	170: //Set the target power to each device
		//Batterys or battery inverters
		//Batterys are only a "normal" Device, when the self consumption mode is active.
		IF eOperationMode = E_OperatingMode_EMS.eSelfConsumption THEN 
			FOR liLPSetPercentPower := 1 TO Constants_Energy.diMaxNumberOfBatteryInverters BY 1 DO
				IF bSurplusAvailable AND Lynus_Standards.GVL_Energy.stDataOfBatteryInverters[diNrOfEMS_OUT,liLPSetPercentPower].byPriority = bySmGrActiveCommonPrio AND Lynus_Standards.GVL_Energy.stDataOfBatteryInverters[diNrOfEMS_OUT,liLPSetPercentPower].rTargetPowerEMS > -100 THEN 
					Lynus_Standards.GVL_Energy.stDataOfBatteryInverters[diNrOfEMS_OUT,liLPSetPercentPower].rTargetPowerEMS := Lynus_Standards.GVL_Energy.stDataOfBatteryInverters[diNrOfEMS_OUT,liLPSetPercentPower].rTargetPowerEMS - rValuePercentToControllableDevices; 
				END_IF
				IF bSurplusAvailable AND Lynus_Standards.GVL_Energy.stDataOfBatteryInverters[diNrOfEMS_OUT,liLPSetPercentPower].rTargetPowerEMS < -100 THEN 
					Lynus_Standards.GVL_Energy.stDataOfBatteryInverters[diNrOfEMS_OUT,liLPSetPercentPower].rTargetPowerEMS := -100; 
				END_IF 
				IF NOT bSurplusAvailable AND Lynus_Standards.GVL_Energy.stDataOfBatteryInverters[diNrOfEMS_OUT,liLPSetPercentPower].byPriority = bySmGrActiveCommonPrio AND Lynus_Standards.GVL_Energy.stDataOfBatteryInverters[diNrOfEMS_OUT,liLPSetPercentPower].rTargetPowerEMS < 0 THEN 
					Lynus_Standards.GVL_Energy.stDataOfBatteryInverters[diNrOfEMS_OUT,liLPSetPercentPower].rTargetPowerEMS := Lynus_Standards.GVL_Energy.stDataOfBatteryInverters[diNrOfEMS_OUT,liLPSetPercentPower].rTargetPowerEMS + rValuePercentToControllableDevices; 
				END_IF
				IF NOT bSurplusAvailable AND Lynus_Standards.GVL_Energy.stDataOfBatteryInverters[diNrOfEMS_OUT,liLPSetPercentPower].rTargetPowerEMS > 0 THEN 
					Lynus_Standards.GVL_Energy.stDataOfBatteryInverters[diNrOfEMS_OUT,liLPSetPercentPower].rTargetPowerEMS := 0; 
				END_IF
				//Power Data is Missing
				IF bMissingPowerData AND Lynus_Standards.GVL_Energy.stDataOfBatteryInverters[diNrOfEMS_OUT,liLPSetPercentPower].byPriority = bySmGrActiveCommonPrio THEN 
					Lynus_Standards.GVL_Energy.stDataOfBatteryInverters[diNrOfEMS_OUT,liLPSetPercentPower].rTargetPowerEMS := 0;	
				END_IF 
				//Limit
				Lynus_Standards.GVL_Energy.stDataOfBatteryInverters[diNrOfEMS_OUT,liLPSetPercentPower].rTargetPowerEMS := LIMIT(-100,Lynus_Standards.GVL_Energy.stDataOfBatteryInverters[diNrOfEMS_OUT,liLPSetPercentPower].rTargetPowerEMS,100);	
			END_FOR
		END_IF
		//Heating pumps
		IF arrActualStepInTurn[1] >= 1 AND arrActualStepInTurn[1] <= 2 THEN
			FOR liLPSetPercentPower := 1 TO Constants_Energy.diMaxNumberOfHeatingPumps BY 1 DO
				//On/Off
				IF bSurplusAvailable AND Lynus_Standards.GVL_Energy.stDataHeatingPumps[diNrOfEMS_OUT,liLPSetPercentPower].byPriority = bySmGrActiveCommonPrio AND Lynus_Standards.GVL_Energy.stDataHeatingPumps[diNrOfEMS_OUT,liLPSetPercentPower].arrTargetPowerEMS[arrActualStepInTurn[1]] < 100 AND NOT 
				Lynus_Standards.GVL_Energy.stDataHeatingPumps[diNrOfEMS_OUT,liLPSetPercentPower].bIsControllable AND NOT Lynus_Standards.GVL_Energy.stDataHeatingPumps[diNrOfEMS_OUT,liLPSetPercentPower].bIsStepSwitched THEN
					Lynus_Standards.GVL_Energy.stDataHeatingPumps[diNrOfEMS_OUT,liLPSetPercentPower].arrTargetPowerEMS[arrActualStepInTurn[1]] := rValuePercentToStepSwitchedDevices; 
				END_IF
				//Controllable linear
				IF bSurplusAvailable AND Lynus_Standards.GVL_Energy.stDataHeatingPumps[diNrOfEMS_OUT,liLPSetPercentPower].byPriority = bySmGrActiveCommonPrio AND Lynus_Standards.GVL_Energy.stDataHeatingPumps[diNrOfEMS_OUT,liLPSetPercentPower].arrTargetPowerEMS[arrActualStepInTurn[1]] < 100 AND 
				Lynus_Standards.GVL_Energy.stDataHeatingPumps[diNrOfEMS_OUT,liLPSetPercentPower].bIsControllable AND NOT Lynus_Standards.GVL_Energy.stDataHeatingPumps[diNrOfEMS_OUT,liLPSetPercentPower].bIsStepSwitched THEN
					Lynus_Standards.GVL_Energy.stDataHeatingPumps[diNrOfEMS_OUT,liLPSetPercentPower].arrTargetPowerEMS[arrActualStepInTurn[1]] := Lynus_Standards.GVL_Energy.stDataHeatingPumps[diNrOfEMS_OUT,liLPSetPercentPower].arrTargetPowerEMS[arrActualStepInTurn[1]] + rValuePercentToControllableDevices; 
				END_IF
				//Step switched
				IF bSurplusAvailable AND Lynus_Standards.GVL_Energy.stDataHeatingPumps[diNrOfEMS_OUT,liLPSetPercentPower].byPriority = bySmGrActiveCommonPrio AND Lynus_Standards.GVL_Energy.stDataHeatingPumps[diNrOfEMS_OUT,liLPSetPercentPower].arrTargetPowerEMS[arrActualStepInTurn[1]] < 100 AND 
				Lynus_Standards.GVL_Energy.stDataHeatingPumps[diNrOfEMS_OUT,liLPSetPercentPower].bIsControllable AND Lynus_Standards.GVL_Energy.stDataHeatingPumps[diNrOfEMS_OUT,liLPSetPercentPower].bIsStepSwitched THEN
					Lynus_Standards.GVL_Energy.stDataHeatingPumps[diNrOfEMS_OUT,liLPSetPercentPower].arrTargetPowerEMS[arrActualStepInTurn[1]] := rValuePercentToStepSwitchedDevices; 
				END_IF
				IF bSurplusAvailable AND Lynus_Standards.GVL_Energy.stDataHeatingPumps[diNrOfEMS_OUT,liLPSetPercentPower].arrTargetPowerEMS[arrActualStepInTurn[1]] > 100 THEN 
					Lynus_Standards.GVL_Energy.stDataHeatingPumps[diNrOfEMS_OUT,liLPSetPercentPower].arrTargetPowerEMS[arrActualStepInTurn[1]] := 100; 
				END_IF 
				//On/Off
				IF NOT bSurplusAvailable AND Lynus_Standards.GVL_Energy.stDataHeatingPumps[diNrOfEMS_OUT,liLPSetPercentPower].byPriority = bySmGrActiveCommonPrio AND Lynus_Standards.GVL_Energy.stDataHeatingPumps[diNrOfEMS_OUT,liLPSetPercentPower].arrTargetPowerEMS[arrActualStepInTurn[1]] > 0 AND NOT 
				Lynus_Standards.GVL_Energy.stDataHeatingPumps[diNrOfEMS_OUT,liLPSetPercentPower].bIsControllable AND NOT Lynus_Standards.GVL_Energy.stDataHeatingPumps[diNrOfEMS_OUT,liLPSetPercentPower].bIsStepSwitched THEN
					Lynus_Standards.GVL_Energy.stDataHeatingPumps[diNrOfEMS_OUT,liLPSetPercentPower].arrTargetPowerEMS[arrActualStepInTurn[1]] := rValuePercentToStepSwitchedDevices; 
				END_IF
				//Controllable linear
				IF NOT bSurplusAvailable AND Lynus_Standards.GVL_Energy.stDataHeatingPumps[diNrOfEMS_OUT,liLPSetPercentPower].byPriority = bySmGrActiveCommonPrio AND Lynus_Standards.GVL_Energy.stDataHeatingPumps[diNrOfEMS_OUT,liLPSetPercentPower].arrTargetPowerEMS[arrActualStepInTurn[1]] > 0 AND 
				Lynus_Standards.GVL_Energy.stDataHeatingPumps[diNrOfEMS_OUT,liLPSetPercentPower].bIsControllable AND NOT Lynus_Standards.GVL_Energy.stDataHeatingPumps[diNrOfEMS_OUT,liLPSetPercentPower].bIsStepSwitched THEN
					Lynus_Standards.GVL_Energy.stDataHeatingPumps[diNrOfEMS_OUT,liLPSetPercentPower].arrTargetPowerEMS[arrActualStepInTurn[1]] := Lynus_Standards.GVL_Energy.stDataHeatingPumps[diNrOfEMS_OUT,liLPSetPercentPower].arrTargetPowerEMS[arrActualStepInTurn[1]] - rValuePercentToControllableDevices; 
				END_IF
				//Step switched
				IF NOT bSurplusAvailable AND Lynus_Standards.GVL_Energy.stDataHeatingPumps[diNrOfEMS_OUT,liLPSetPercentPower].byPriority = bySmGrActiveCommonPrio AND Lynus_Standards.GVL_Energy.stDataHeatingPumps[diNrOfEMS_OUT,liLPSetPercentPower].arrTargetPowerEMS[arrActualStepInTurn[1]] > 0 AND 
				Lynus_Standards.GVL_Energy.stDataHeatingPumps[diNrOfEMS_OUT,liLPSetPercentPower].bIsControllable AND Lynus_Standards.GVL_Energy.stDataHeatingPumps[diNrOfEMS_OUT,liLPSetPercentPower].bIsStepSwitched THEN
					Lynus_Standards.GVL_Energy.stDataHeatingPumps[diNrOfEMS_OUT,liLPSetPercentPower].arrTargetPowerEMS[arrActualStepInTurn[1]] := rValuePercentToStepSwitchedDevices; 
				END_IF
				IF NOT bSurplusAvailable AND Lynus_Standards.GVL_Energy.stDataHeatingPumps[diNrOfEMS_OUT,liLPSetPercentPower].arrTargetPowerEMS[arrActualStepInTurn[1]] < 0 THEN 
					Lynus_Standards.GVL_Energy.stDataHeatingPumps[diNrOfEMS_OUT,liLPSetPercentPower].arrTargetPowerEMS[arrActualStepInTurn[1]] := 0; 
				END_IF
				//Limit
				Lynus_Standards.GVL_Energy.stDataHeatingPumps[diNrOfEMS_OUT,liLPSetPercentPower].arrTargetPowerEMS[arrActualStepInTurn[1]] := LIMIT(0,Lynus_Standards.GVL_Energy.stDataHeatingPumps[diNrOfEMS_OUT,liLPSetPercentPower].arrTargetPowerEMS[arrActualStepInTurn[1]],100);
			END_FOR
		END_IF
		//electric heating element
		IF arrActualStepInTurn[2] >= 1 AND arrActualStepInTurn[2] <= 10 THEN
			FOR liLPSetPercentPower := 1 TO Constants_Energy.diMaxNumberOfElectricHeatingElements BY 1 DO
				//On/Off
				IF bSurplusAvailable AND Lynus_Standards.GVL_Energy.stDataElectricHeatingElements[diNrOfEMS_OUT,liLPSetPercentPower].byPriority = bySmGrActiveCommonPrio AND Lynus_Standards.GVL_Energy.stDataElectricHeatingElements[diNrOfEMS_OUT,liLPSetPercentPower].arrTargetPowerEMS[arrActualStepInTurn[2]] < 100 AND NOT
				Lynus_Standards.GVL_Energy.stDataElectricHeatingElements[diNrOfEMS_OUT,liLPSetPercentPower].bIsControllable AND NOT Lynus_Standards.GVL_Energy.stDataElectricHeatingElements[diNrOfEMS_OUT,liLPSetPercentPower].bIsStepSwitched THEN
					Lynus_Standards.GVL_Energy.stDataElectricHeatingElements[diNrOfEMS_OUT,liLPSetPercentPower].arrTargetPowerEMS[arrActualStepInTurn[2]] := rValuePercentToStepSwitchedDevices;
				END_IF
				//Controllable linear
				IF bSurplusAvailable AND Lynus_Standards.GVL_Energy.stDataElectricHeatingElements[diNrOfEMS_OUT,liLPSetPercentPower].byPriority = bySmGrActiveCommonPrio AND Lynus_Standards.GVL_Energy.stDataElectricHeatingElements[diNrOfEMS_OUT,liLPSetPercentPower].arrTargetPowerEMS[arrActualStepInTurn[2]] < 100 AND
				Lynus_Standards.GVL_Energy.stDataElectricHeatingElements[diNrOfEMS_OUT,liLPSetPercentPower].bIsControllable AND NOT Lynus_Standards.GVL_Energy.stDataElectricHeatingElements[diNrOfEMS_OUT,liLPSetPercentPower].bIsStepSwitched THEN
					Lynus_Standards.GVL_Energy.stDataElectricHeatingElements[diNrOfEMS_OUT,liLPSetPercentPower].arrTargetPowerEMS[arrActualStepInTurn[2]] := Lynus_Standards.GVL_Energy.stDataElectricHeatingElements[diNrOfEMS_OUT,liLPSetPercentPower].arrTargetPowerEMS[arrActualStepInTurn[2]] + rValuePercentToControllableDevices;
				END_IF
				//Step switched
				IF bSurplusAvailable AND Lynus_Standards.GVL_Energy.stDataElectricHeatingElements[diNrOfEMS_OUT,liLPSetPercentPower].byPriority = bySmGrActiveCommonPrio AND Lynus_Standards.GVL_Energy.stDataElectricHeatingElements[diNrOfEMS_OUT,liLPSetPercentPower].arrTargetPowerEMS[arrActualStepInTurn[2]] < 100 AND
				Lynus_Standards.GVL_Energy.stDataElectricHeatingElements[diNrOfEMS_OUT,liLPSetPercentPower].bIsControllable AND Lynus_Standards.GVL_Energy.stDataElectricHeatingElements[diNrOfEMS_OUT,liLPSetPercentPower].bIsStepSwitched THEN
					Lynus_Standards.GVL_Energy.stDataElectricHeatingElements[diNrOfEMS_OUT,liLPSetPercentPower].arrTargetPowerEMS[arrActualStepInTurn[2]] := rValuePercentToStepSwitchedDevices;
				END_IF
				IF bSurplusAvailable AND Lynus_Standards.GVL_Energy.stDataElectricHeatingElements[diNrOfEMS_OUT,liLPSetPercentPower].arrTargetPowerEMS[arrActualStepInTurn[2]] > 100 THEN 
					Lynus_Standards.GVL_Energy.stDataElectricHeatingElements[diNrOfEMS_OUT,liLPSetPercentPower].arrTargetPowerEMS[arrActualStepInTurn[2]] := 100; 
				END_IF
				//On/Off
				IF NOT bSurplusAvailable AND Lynus_Standards.GVL_Energy.stDataElectricHeatingElements[diNrOfEMS_OUT,liLPSetPercentPower].byPriority = bySmGrActiveCommonPrio AND Lynus_Standards.GVL_Energy.stDataElectricHeatingElements[diNrOfEMS_OUT,liLPSetPercentPower].arrTargetPowerEMS[arrActualStepInTurn[2]] > 0 AND NOT
				Lynus_Standards.GVL_Energy.stDataElectricHeatingElements[diNrOfEMS_OUT,liLPSetPercentPower].bIsControllable AND NOT Lynus_Standards.GVL_Energy.stDataElectricHeatingElements[diNrOfEMS_OUT,liLPSetPercentPower].bIsStepSwitched THEN
					Lynus_Standards.GVL_Energy.stDataElectricHeatingElements[diNrOfEMS_OUT,liLPSetPercentPower].arrTargetPowerEMS[arrActualStepInTurn[2]] := rValuePercentToStepSwitchedDevices;
				END_IF
				//Controllable linear
				IF NOT bSurplusAvailable AND Lynus_Standards.GVL_Energy.stDataElectricHeatingElements[diNrOfEMS_OUT,liLPSetPercentPower].byPriority = bySmGrActiveCommonPrio AND Lynus_Standards.GVL_Energy.stDataElectricHeatingElements[diNrOfEMS_OUT,liLPSetPercentPower].arrTargetPowerEMS[arrActualStepInTurn[2]] > 0 AND
				Lynus_Standards.GVL_Energy.stDataElectricHeatingElements[diNrOfEMS_OUT,liLPSetPercentPower].bIsControllable AND NOT Lynus_Standards.GVL_Energy.stDataElectricHeatingElements[diNrOfEMS_OUT,liLPSetPercentPower].bIsStepSwitched THEN
					Lynus_Standards.GVL_Energy.stDataElectricHeatingElements[diNrOfEMS_OUT,liLPSetPercentPower].arrTargetPowerEMS[arrActualStepInTurn[2]] := Lynus_Standards.GVL_Energy.stDataElectricHeatingElements[diNrOfEMS_OUT,liLPSetPercentPower].arrTargetPowerEMS[arrActualStepInTurn[2]] - rValuePercentToControllableDevices;
				END_IF
				//Step switched
				IF NOT bSurplusAvailable AND Lynus_Standards.GVL_Energy.stDataElectricHeatingElements[diNrOfEMS_OUT,liLPSetPercentPower].byPriority = bySmGrActiveCommonPrio AND Lynus_Standards.GVL_Energy.stDataElectricHeatingElements[diNrOfEMS_OUT,liLPSetPercentPower].arrTargetPowerEMS[arrActualStepInTurn[2]] > 0 AND
				Lynus_Standards.GVL_Energy.stDataElectricHeatingElements[diNrOfEMS_OUT,liLPSetPercentPower].bIsControllable AND Lynus_Standards.GVL_Energy.stDataElectricHeatingElements[diNrOfEMS_OUT,liLPSetPercentPower].bIsStepSwitched THEN
					Lynus_Standards.GVL_Energy.stDataElectricHeatingElements[diNrOfEMS_OUT,liLPSetPercentPower].arrTargetPowerEMS[arrActualStepInTurn[2]] := rValuePercentToStepSwitchedDevices;
				END_IF	
				IF NOT bSurplusAvailable AND Lynus_Standards.GVL_Energy.stDataElectricHeatingElements[diNrOfEMS_OUT,liLPSetPercentPower].arrTargetPowerEMS[arrActualStepInTurn[2]] < 0 THEN 
					Lynus_Standards.GVL_Energy.stDataElectricHeatingElements[diNrOfEMS_OUT,liLPSetPercentPower].arrTargetPowerEMS[arrActualStepInTurn[2]] := 0; 
				END_IF 
				//Limit
				Lynus_Standards.GVL_Energy.stDataElectricHeatingElements[diNrOfEMS_OUT,liLPSetPercentPower].arrTargetPowerEMS[arrActualStepInTurn[2]] := LIMIT(0,Lynus_Standards.GVL_Energy.stDataElectricHeatingElements[diNrOfEMS_OUT,liLPSetPercentPower].arrTargetPowerEMS[arrActualStepInTurn[2]],100);
			END_FOR			
		END_IF
		//Other big consumer
		FOR liLPSetPercentPower := 1 TO Constants_Energy.diMaxNumberOfOtherBigConsumers BY 1 DO
			//On/Off
			IF bSurplusAvailable AND Lynus_Standards.GVL_Energy.stDataOtherBigConsumers[diNrOfEMS_OUT,liLPSetPercentPower].byPriority = bySmGrActiveCommonPrio AND Lynus_Standards.GVL_Energy.stDataOtherBigConsumers[diNrOfEMS_OUT,liLPSetPercentPower].rTargetPowerEMS < 100 AND NOT
			Lynus_Standards.GVL_Energy.stDataOtherBigConsumers[diNrOfEMS_OUT,liLPSetPercentPower].bIsControllable THEN 
				Lynus_Standards.GVL_Energy.stDataOtherBigConsumers[diNrOfEMS_OUT,liLPSetPercentPower].rTargetPowerEMS := rValuePercentToStepSwitchedDevices; 
			END_IF
			//Controllable linear
			IF bSurplusAvailable AND Lynus_Standards.GVL_Energy.stDataOtherBigConsumers[diNrOfEMS_OUT,liLPSetPercentPower].byPriority = bySmGrActiveCommonPrio AND Lynus_Standards.GVL_Energy.stDataOtherBigConsumers[diNrOfEMS_OUT,liLPSetPercentPower].rTargetPowerEMS < 100 AND
			Lynus_Standards.GVL_Energy.stDataOtherBigConsumers[diNrOfEMS_OUT,liLPSetPercentPower].bIsControllable THEN 
				Lynus_Standards.GVL_Energy.stDataOtherBigConsumers[diNrOfEMS_OUT,liLPSetPercentPower].rTargetPowerEMS := Lynus_Standards.GVL_Energy.stDataOtherBigConsumers[diNrOfEMS_OUT,liLPSetPercentPower].rTargetPowerEMS + rValuePercentToControllableDevices;
			END_IF
			IF bSurplusAvailable AND Lynus_Standards.GVL_Energy.stDataOtherBigConsumers[diNrOfEMS_OUT,liLPSetPercentPower].rTargetPowerEMS > 100 THEN 
				Lynus_Standards.GVL_Energy.stDataOtherBigConsumers[diNrOfEMS_OUT,liLPSetPercentPower].rTargetPowerEMS := 100; 
			END_IF
			//On/Off
			IF NOT bSurplusAvailable AND Lynus_Standards.GVL_Energy.stDataOtherBigConsumers[diNrOfEMS_OUT,liLPSetPercentPower].byPriority = bySmGrActiveCommonPrio AND Lynus_Standards.GVL_Energy.stDataOtherBigConsumers[diNrOfEMS_OUT,liLPSetPercentPower].rTargetPowerEMS > 0 AND NOT
				Lynus_Standards.GVL_Energy.stDataOtherBigConsumers[diNrOfEMS_OUT,liLPSetPercentPower].bIsControllable THEN Lynus_Standards.GVL_Energy.stDataOtherBigConsumers[diNrOfEMS_OUT,liLPSetPercentPower].rTargetPowerEMS := rValuePercentToStepSwitchedDevices; 
			END_IF
			//Controllable linear
			IF NOT bSurplusAvailable AND Lynus_Standards.GVL_Energy.stDataOtherBigConsumers[diNrOfEMS_OUT,liLPSetPercentPower].byPriority = bySmGrActiveCommonPrio AND Lynus_Standards.GVL_Energy.stDataOtherBigConsumers[diNrOfEMS_OUT,liLPSetPercentPower].rTargetPowerEMS > 0 AND
			Lynus_Standards.GVL_Energy.stDataOtherBigConsumers[diNrOfEMS_OUT,liLPSetPercentPower].bIsControllable THEN 
				Lynus_Standards.GVL_Energy.stDataOtherBigConsumers[diNrOfEMS_OUT,liLPSetPercentPower].rTargetPowerEMS := Lynus_Standards.GVL_Energy.stDataOtherBigConsumers[diNrOfEMS_OUT,liLPSetPercentPower].rTargetPowerEMS - rValuePercentToControllableDevices;
			END_IF
			IF NOT bSurplusAvailable AND Lynus_Standards.GVL_Energy.stDataOtherBigConsumers[diNrOfEMS_OUT,liLPSetPercentPower].rTargetPowerEMS < 0 THEN 
				Lynus_Standards.GVL_Energy.stDataOtherBigConsumers[diNrOfEMS_OUT,liLPSetPercentPower].rTargetPowerEMS := 0; 
			END_IF
			//Limit
			Lynus_Standards.GVL_Energy.stDataOtherBigConsumers[diNrOfEMS_OUT,liLPSetPercentPower].rTargetPowerEMS := LIMIT(0,Lynus_Standards.GVL_Energy.stDataOtherBigConsumers[diNrOfEMS_OUT,liLPSetPercentPower].rTargetPowerEMS,100);
		END_FOR
		//Electric charging stations
		FOR liLPSetPercentPower := 1 TO Constants_Energy.diMaxNumberOfElectricChargingStations BY 1 DO
			//On/Off
			IF bSurplusAvailable AND Lynus_Standards.GVL_Energy.stDataElectricChargingStations[diNrOfEMS_OUT,liLPSetPercentPower].byPriority = bySmGrActiveCommonPrio AND Lynus_Standards.GVL_Energy.stDataElectricChargingStations[diNrOfEMS_OUT,liLPSetPercentPower].rTargetPowerEMS < 100 AND NOT 
			Lynus_Standards.GVL_Energy.stDataElectricChargingStations[diNrOfEMS_OUT,liLPSetPercentPower].bIsControllable THEN 
				//No power on ECS because on the Electric Fuse Line we take to much Power on witch the ECS is conected
				IF NOT bNoPowerForECS THEN 
					Lynus_Standards.GVL_Energy.stDataElectricChargingStations[diNrOfEMS_OUT,liLPSetPercentPower].rTargetPowerEMS := rValuePercentToStepSwitchedDevices;	
				END_IF	
			END_IF
			//Controllable linear
			IF bSurplusAvailable AND Lynus_Standards.GVL_Energy.stDataElectricChargingStations[diNrOfEMS_OUT,liLPSetPercentPower].byPriority = bySmGrActiveCommonPrio AND Lynus_Standards.GVL_Energy.stDataElectricChargingStations[diNrOfEMS_OUT,liLPSetPercentPower].rTargetPowerEMS < 100 AND 
			Lynus_Standards.GVL_Energy.stDataElectricChargingStations[diNrOfEMS_OUT,liLPSetPercentPower].bIsControllable THEN 
				//No power on ECS because on the Electric Fuse Line we take to much Power on witch the ECS is conected
				IF NOT bNoPowerForECS THEN
					Lynus_Standards.GVL_Energy.stDataElectricChargingStations[diNrOfEMS_OUT,liLPSetPercentPower].rTargetPowerEMS := Lynus_Standards.GVL_Energy.stDataElectricChargingStations[diNrOfEMS_OUT,liLPSetPercentPower].rTargetPowerEMS + rValuePercentToControllableDevices;		
				END_IF
			END_IF
			IF bSurplusAvailable AND Lynus_Standards.GVL_Energy.stDataElectricChargingStations[diNrOfEMS_OUT,liLPSetPercentPower].rTargetPowerEMS > 100 THEN 
				Lynus_Standards.GVL_Energy.stDataElectricChargingStations[diNrOfEMS_OUT,liLPSetPercentPower].rTargetPowerEMS := 100; 
			END_IF
			//On/Off
			IF NOT bSurplusAvailable AND Lynus_Standards.GVL_Energy.stDataElectricChargingStations[diNrOfEMS_OUT,liLPSetPercentPower].byPriority = bySmGrActiveCommonPrio AND Lynus_Standards.GVL_Energy.stDataElectricChargingStations[diNrOfEMS_OUT,liLPSetPercentPower].rTargetPowerEMS > 0 AND NOT 
			Lynus_Standards.GVL_Energy.stDataElectricChargingStations[diNrOfEMS_OUT,liLPSetPercentPower].bIsControllable THEN 
				Lynus_Standards.GVL_Energy.stDataElectricChargingStations[diNrOfEMS_OUT,liLPSetPercentPower].rTargetPowerEMS := rValuePercentToStepSwitchedDevices;		
			END_IF
			//Controllable linear
			IF NOT bSurplusAvailable AND Lynus_Standards.GVL_Energy.stDataElectricChargingStations[diNrOfEMS_OUT,liLPSetPercentPower].byPriority = bySmGrActiveCommonPrio AND Lynus_Standards.GVL_Energy.stDataElectricChargingStations[diNrOfEMS_OUT,liLPSetPercentPower].rTargetPowerEMS > 0 AND 
			Lynus_Standards.GVL_Energy.stDataElectricChargingStations[diNrOfEMS_OUT,liLPSetPercentPower].bIsControllable THEN 
				Lynus_Standards.GVL_Energy.stDataElectricChargingStations[diNrOfEMS_OUT,liLPSetPercentPower].rTargetPowerEMS := Lynus_Standards.GVL_Energy.stDataElectricChargingStations[diNrOfEMS_OUT,liLPSetPercentPower].rTargetPowerEMS - rValuePercentToControllableDevices;	
			END_IF
			IF NOT bSurplusAvailable AND Lynus_Standards.GVL_Energy.stDataElectricChargingStations[diNrOfEMS_OUT,liLPSetPercentPower].rTargetPowerEMS < 0 THEN 
				Lynus_Standards.GVL_Energy.stDataElectricChargingStations[diNrOfEMS_OUT,liLPSetPercentPower].rTargetPowerEMS := 0; 
			END_IF	
			//Limit
			Lynus_Standards.GVL_Energy.stDataElectricChargingStations[diNrOfEMS_OUT,liLPSetPercentPower].rTargetPowerEMS := LIMIT(0,Lynus_Standards.GVL_Energy.stDataElectricChargingStations[diNrOfEMS_OUT,liLPSetPercentPower].rTargetPowerEMS,100);
		END_FOR 
		uiState := 10;
END_CASE

(*-------------------------------------------------------------------------------------Correction Charging stations regarding max fuse power---------------------------------------------------------------------------------------------------------------*)

//Correction for the charging station power that the target power is not bigger then the maximum of the fuse. Active on mode peak load capping (Index from meter > 0 and fuse value > 0) and load management (always).
//Work only with controllable charging station. Not work for On/off stations.
IF (stSetupEMS.bEnableMainFuseFunction AND bEnable AND (eOperationMode = E_OperatingMode_EMS.ePeakLoadCapping OR eOperationMode = E_OperatingMode_EMS.eLoadManagement)) THEN
	IF arrMaxPrioReached[5] THEN 
		bECSPrio255 := TRUE; 
	END_IF
	IF NOT bSurplusAvailable THEN 
		bECSPrio255 := FALSE; 
	END_IF

	lrPowerDiffFuseECS := (stSetupEMS.rSizeMainFuseCS * 0.95) - Lynus_Standards.GVL_Energy.stDataElectricMeters[diNrOfEM_IN_ECS].lrPowerConsumption;	
	//Make little tolerance that we dont regulate up and down 
	IF lrPowerDiffFuseECS > 0 AND lrPowerDiffFuseECS <= 0.1 THEN 
		lrPowerDiffFuseECS := 0; 
	END_IF  
	IF lrPowerDiffFuseECS > 0 THEN 
		lrPowerDiffFuseECS := lrPowerDiffFuseECS - 0.1; 
	END_IF 
	
	//No power for ECS on normal EMS Step
	IF lrPowerDiffFuseECS < 0 THEN 
		bNoPowerForECS := TRUE; 
	ELSE
		bNoPowerForECS := FALSE;
	END_IF	
		
	diNumberOfECS := 0;		
	FOR liLPCorrectionPowerCS := 1 TO Constants_Energy.diMaxNumberOfElectricChargingStations BY 1 DO
		//Count number of charging stations when we have surplus on Fuse Line
		IF NOT arrMinPrioReached[5] AND Lynus_Standards.GVL_Energy.stDataElectricChargingStations[diNrOfEMS_OUT,liLPCorrectionPowerCS].byPriority <= bySmGrActiveCommonPrio AND 
			Lynus_Standards.GVL_Energy.stDataElectricChargingStations[diNrOfEMS_OUT,liLPCorrectionPowerCS].bEnabled AND 
			Lynus_Standards.GVL_Energy.stDataElectricChargingStations[diNrOfEMS_OUT,liLPCorrectionPowerCS].rTargetPowerEMS < 100 AND lrPowerDiffFuseECS >= 0 THEN 
			diNumberOfECS := diNumberOfECS + 1; 
		END_IF
		//Count number of charging stations when we have NO surplus on Fuse Line
		IF NOT arrMinPrioReached[5] AND Lynus_Standards.GVL_Energy.stDataElectricChargingStations[diNrOfEMS_OUT,liLPCorrectionPowerCS].byPriority <= bySmGrActiveCommonPrio AND 
		Lynus_Standards.GVL_Energy.stDataElectricChargingStations[diNrOfEMS_OUT,liLPCorrectionPowerCS].bEnabled AND
		Lynus_Standards.GVL_Energy.stDataElectricChargingStations[diNrOfEMS_OUT,liLPCorrectionPowerCS].rTargetPowerEMS > 0 AND lrPowerDiffFuseECS < 0 THEN 
			diNumberOfECS := diNumberOfECS + 1; 
		END_IF 
	END_FOR
	//Calculate the power in % for each charging station
	//Actual Power is <= then stSetupEMS.rSizeMainFuseCS 
	IF diNumberOfECS > 0 AND lrPowerDiffFuseECS >= 0 THEN 
		lrPowerForCalculateECS := lrPowerDiffFuseECS / diNumberOfECS; 
	END_IF  
	//Actual Power is > then stSetupEMS.rSizeMainFuseCS
	IF diNumberOfECS > 0 AND lrPowerDiffFuseECS < 0 THEN 
		lrPowerForCalculateECS := (lrPowerDiffFuseECS * - 1) / diNumberOfECS; 
	END_IF 

	//Timer to make the correction for the charging stations
	IF (NOT arrMinPrioReached[5] AND NOT timCorrectionECS.Q AND bEnable AND (eOperationMode = E_OperatingMode_EMS.ePeakLoadCapping OR eOperationMode = E_OperatingMode_EMS.eLoadManagement)) THEN  
		timCorrectionECS.IN := TRUE;
	ELSE
		timCorrectionECS.IN := FALSE;
	END_IF
	//The timer work faster when the value from lrPowerDiffFuseECS is bigger
	//Positive value (Mean more power for ECS)
	IF lrPowerDiffFuseECS >= 0.75 THEN 
		timCorrectionECS.PT := T#2.5S; 
	END_IF
	IF lrPowerDiffFuseECS >= 0.5 AND lrPowerDiffFuseECS < 0.75 THEN 
		timCorrectionECS.PT := T#3S; 
	END_IF
	IF lrPowerDiffFuseECS >= 0.25 AND lrPowerDiffFuseECS < 0.5 THEN 
		timCorrectionECS.PT := T#3.5S; 
	END_IF
	IF lrPowerDiffFuseECS > 0 AND lrPowerDiffFuseECS < 0.25 THEN 
		timCorrectionECS.PT := T#4S; 
	END_IF
	//Value is 0
	IF lrPowerDiffFuseECS = 0 THEN 
		timCorrectionECS.PT := T#5S; 
	END_IF 
	//Negative value (Mean less power for ECS)
	IF lrPowerDiffFuseECS < 0 AND lrPowerDiffFuseECS > - 0.25 
		THEN timCorrectionECS.PT := T#4S; 
	END_IF
	IF lrPowerDiffFuseECS <= - 0.25 AND lrPowerDiffFuseECS > - 0.5 THEN 
		timCorrectionECS.PT := T#3.5S; 
	END_IF
	IF lrPowerDiffFuseECS <= - 0.5 AND lrPowerDiffFuseECS > - 0.75 THEN 
		timCorrectionECS.PT := T#3S; 
	END_IF
	IF lrPowerDiffFuseECS <= - 0.75 THEN 
		timCorrectionECS.PT := T#2.5S; 
	END_IF
	//Timer
	timCorrectionECS(IN:= , PT:= , Q=> , ET=> );				
			
//Set the new power to the charging stations with priority < common priority in progress
	lrTargetPowerCorrectionECS := 0;
	FOR liLPCorrectionPowerCS := 1 TO Constants_Energy.diMaxNumberOfElectricChargingStations BY 1 DO 	
		IF (NOT arrMinPrioReached[5] AND timCorrectionECS.Q AND Lynus_Standards.GVL_Energy.stDataElectricChargingStations[diNrOfEMS_OUT,liLPCorrectionPowerCS].byPriority < bySmGrActiveCommonPrio AND eOperationMode = E_OperatingMode_EMS.ePeakLoadCapping AND stSetupEMS.rSizeMainFuseCS > 0 AND Lynus_Standards.GVL_Energy.stDataElectricMeters[diNrOfEM_IN_ECS].bEnabled) OR
		(NOT arrMinPrioReached[5] AND timCorrectionECS.Q AND Lynus_Standards.GVL_Energy.stDataElectricChargingStations[diNrOfEMS_OUT,liLPCorrectionPowerCS].byPriority < bySmGrActiveCommonPrio AND eOperationMode = E_OperatingMode_EMS.eLoadManagement AND stSetupEMS.rSizeMainFuseCS > 0 AND Lynus_Standards.GVL_Energy.stDataElectricMeters[diNrOfEM_IN_ECS].bEnabled) OR
		(NOT arrMinPrioReached[5] AND timCorrectionECS.Q AND lrPowerDiffFuseECS < 0 AND Lynus_Standards.GVL_Energy.stDataElectricChargingStations[diNrOfEMS_OUT,liLPCorrectionPowerCS].byPriority = bySmGrActiveCommonPrio AND eOperationMode = E_OperatingMode_EMS.ePeakLoadCapping AND stSetupEMS.rSizeMainFuseCS > 0 AND Lynus_Standards.GVL_Energy.stDataElectricMeters[diNrOfEM_IN_ECS].bEnabled) OR
		(NOT arrMinPrioReached[5] AND timCorrectionECS.Q AND lrPowerDiffFuseECS < 0 AND Lynus_Standards.GVL_Energy.stDataElectricChargingStations[diNrOfEMS_OUT,liLPCorrectionPowerCS].byPriority = bySmGrActiveCommonPrio AND eOperationMode = E_OperatingMode_EMS.eLoadManagement AND stSetupEMS.rSizeMainFuseCS > 0 AND Lynus_Standards.GVL_Energy.stDataElectricMeters[diNrOfEM_IN_ECS].bEnabled) OR				
		(NOT arrMinPrioReached[5] AND timCorrectionECS.Q AND Lynus_Standards.GVL_Energy.stDataElectricChargingStations[diNrOfEMS_OUT,liLPCorrectionPowerCS].byPriority = 255 AND bECSPrio255 AND eOperationMode = E_OperatingMode_EMS.ePeakLoadCapping AND stSetupEMS.rSizeMainFuseCS > 0 AND Lynus_Standards.GVL_Energy.stDataElectricMeters[diNrOfEM_IN_ECS].bEnabled) OR	
		(NOT arrMinPrioReached[5] AND timCorrectionECS.Q AND Lynus_Standards.GVL_Energy.stDataElectricChargingStations[diNrOfEMS_OUT,liLPCorrectionPowerCS].byPriority = 255 AND bECSPrio255 AND eOperationMode = E_OperatingMode_EMS.eLoadManagement AND stSetupEMS.rSizeMainFuseCS > 0 AND Lynus_Standards.GVL_Energy.stDataElectricMeters[diNrOfEM_IN_ECS].bEnabled) THEN
			//Calcualte the new % value for each charging station	
			IF Lynus_Standards.GVL_Energy.stDataElectricChargingStations[diNrOfEMS_OUT,liLPCorrectionPowerCS].rMaxPower > 0 THEN 
				lrTargetPowerCorrectionECS := (100 * lrPowerForCalculateECS) / Lynus_Standards.GVL_Energy.stDataElectricChargingStations[diNrOfEMS_OUT,liLPCorrectionPowerCS].rMaxPower;	
				lrTargetPowerCorrectionECS := LIMIT(0,lrTargetPowerCorrectionECS,100);
			ELSE
				//Without power data on the setups from the charging station set target powert to -100 or +100 to dissable the charging station
				IF lrPowerDiffFuseECS >= 0 THEN 
					lrTargetPowerCorrectionECS := - 100; 
				ELSE 
					lrTargetPowerCorrectionECS := 100; 
				END_IF 
			END_IF	
			IF lrPowerDiffFuseECS >= 0 AND Lynus_Standards.GVL_Energy.stDataElectricChargingStations[diNrOfEMS_OUT,liLPCorrectionPowerCS].bIsControllable THEN 
				Lynus_Standards.GVL_Energy.stDataElectricChargingStations[diNrOfEMS_OUT,liLPCorrectionPowerCS].rTargetPowerEMS := Lynus_Standards.GVL_Energy.stDataElectricChargingStations[diNrOfEMS_OUT,liLPCorrectionPowerCS].rTargetPowerEMS + LREAL_TO_REAL(lrTargetPowerCorrectionECS); 
			END_IF
			IF lrPowerDiffFuseECS < 0 AND Lynus_Standards.GVL_Energy.stDataElectricChargingStations[diNrOfEMS_OUT,liLPCorrectionPowerCS].bIsControllable THEN 
				Lynus_Standards.GVL_Energy.stDataElectricChargingStations[diNrOfEMS_OUT,liLPCorrectionPowerCS].rTargetPowerEMS := Lynus_Standards.GVL_Energy.stDataElectricChargingStations[diNrOfEMS_OUT,liLPCorrectionPowerCS].rTargetPowerEMS - LREAL_TO_REAL(lrTargetPowerCorrectionECS); 
			END_IF	
			//Limits
			Lynus_Standards.GVL_Energy.stDataElectricChargingStations[diNrOfEMS_OUT,liLPCorrectionPowerCS].rTargetPowerEMS := LIMIT(0,Lynus_Standards.GVL_Energy.stDataElectricChargingStations[diNrOfEMS_OUT,liLPCorrectionPowerCS].rTargetPowerEMS,100);			
		END_IF
	END_FOR

	//Dissable the ECS complete when the EM has a Error
	IF (Lynus_Standards.GVL_Energy.stDataElectricMeters[diNrOfEM_IN_ECS].byErrorWarning = 2 AND (eOperationMode = E_OperatingMode_EMS.eLoadManagement OR eOperationMode = E_OperatingMode_EMS.ePeakLoadCapping)) THEN
		timResetDisableECS.IN := TRUE;
	ELSE
		timResetDisableECS.IN := FALSE;
	END_IF
	timResetDisableECS(IN:= , PT:= T#10S, Q=> , ET=> );	
	IF timResetDisableECS.Q THEN 
		bDisableECS := TRUE; 
	ELSE 
		bDisableECS := FALSE; 
	END_IF

ELSE
	timResetDisableECS.IN := FALSE;
	bDisableECS := FALSE;		
	timCorrectionECS.IN := FALSE;
	bECSPrio255 := FALSE;
	bNoPowerForECS := FALSE;
END_IF		
		
(*-------------------------------------------------------------------------------------Set the power to 0 on each device---------------------------------------------------------------------------------------------------------------*)	
	
//When a device has the priority 0, the priority is bigger then who was at the moment in progress, the EMS function is not enabled, a positv or negative edge came when the emergency power mode start or stop or when the operation mode is changing then the EMS start from new and all devices are set to defaul target power 0.
//Set the target power to 0 where there should no power 

FPEPO(CLK:= bEPMActive, Q=> );
FNEPO(CLK:= bEPMActive, Q=> );
	
diMemCmpOperationState := MEMCMP(ADR(eOperationMode),ADR(eOperationModeEMS_CP),SIZEOF(eOperationModeEMS_CP)); 	

//Battery	
FOR arrLPPrioZeroSetToZeroP[1] := 1 TO Constants_Energy.diMaxNumberOfBatteryInverters BY 1 DO
	IF Lynus_Standards.GVL_Energy.stDataOfBatteryInverters[diNrOfEMS_OUT,arrLPPrioZeroSetToZeroP[1]].byPriority = 0 OR Lynus_Standards.GVL_Energy.stDataOfBatteryInverters[diNrOfEMS_OUT,arrLPPrioZeroSetToZeroP[1]].byPriority > arrActualPrioInTurn[1] OR arrMinPrioReached[1] OR NOT bEnable OR FPEPO.Q OR FNEPO.Q OR 
		diMemCmpOperationState <> 0 OR eOperationMode = E_OperatingMode_EMS.eAllOff OR bStopAll THEN 
		Lynus_Standards.GVL_Energy.stDataOfBatteryInverters[diNrOfEMS_OUT,arrLPPrioZeroSetToZeroP[1]].rTargetPowerEMS := 0; 
	END_IF
END_FOR
//Heating Pumps
FOR arrLPPrioZeroSetToZeroP[2] := 1 TO Constants_Energy.diMaxNumberOfHeatingPumps BY 1 DO
	IF Lynus_Standards.GVL_Energy.stDataHeatingPumps[diNrOfEMS_OUT,arrLPPrioZeroSetToZeroP[2]].byPriority = 0 OR Lynus_Standards.GVL_Energy.stDataHeatingPumps[diNrOfEMS_OUT,arrLPPrioZeroSetToZeroP[2]].byPriority > arrActualPrioInTurn[2] OR arrMinPrioReached[2] OR NOT bEnable OR FPEPO.Q OR FNEPO.Q OR 
	diMemCmpOperationState <> 0 OR eOperationMode = E_OperatingMode_EMS.eAllOff OR bStopAll THEN
		Lynus_Standards.GVL_Energy.stDataHeatingPumps[diNrOfEMS_OUT,arrLPPrioZeroSetToZeroP[2]].arrTargetPowerEMS[1] := 0;
		Lynus_Standards.GVL_Energy.stDataHeatingPumps[diNrOfEMS_OUT,arrLPPrioZeroSetToZeroP[2]].arrTargetPowerEMS[2] := 0;
		//Switch off external on command for heating pumps
		Lynus_Standards.GVL_Energy.stDataHeatingPumps[diNrOfEMS_OUT,arrLPPrioZeroSetToZeroP[2]].bExternalOnCommand := FALSE;
	END_IF
END_FOR
//EHE
FOR arrLPPrioZeroSetToZeroP[3] := 1 TO Constants_Energy.diMaxNumberOfElectricHeatingElements BY 1 DO
	IF Lynus_Standards.GVL_Energy.stDataElectricHeatingElements[diNrOfEMS_OUT,arrLPPrioZeroSetToZeroP[3]].byPriority = 0 OR Lynus_Standards.GVL_Energy.stDataElectricHeatingElements[diNrOfEMS_OUT,arrLPPrioZeroSetToZeroP[3]].byPriority > arrActualPrioInTurn[3] OR arrMinPrioReached[3] OR NOT bEnable OR FPEPO.Q OR FNEPO.Q OR 
		diMemCmpOperationState <> 0 OR eOperationMode = E_OperatingMode_EMS.eAllOff OR bStopAll THEN 
		Lynus_Standards.GVL_Energy.stDataElectricHeatingElements[diNrOfEMS_OUT,arrLPPrioZeroSetToZeroP[3]].arrTargetPowerEMS[1] := 0;
		Lynus_Standards.GVL_Energy.stDataElectricHeatingElements[diNrOfEMS_OUT,arrLPPrioZeroSetToZeroP[3]].arrTargetPowerEMS[2] := 0;
		Lynus_Standards.GVL_Energy.stDataElectricHeatingElements[diNrOfEMS_OUT,arrLPPrioZeroSetToZeroP[3]].arrTargetPowerEMS[3] := 0;
		Lynus_Standards.GVL_Energy.stDataElectricHeatingElements[diNrOfEMS_OUT,arrLPPrioZeroSetToZeroP[3]].arrTargetPowerEMS[4] := 0;
		Lynus_Standards.GVL_Energy.stDataElectricHeatingElements[diNrOfEMS_OUT,arrLPPrioZeroSetToZeroP[3]].arrTargetPowerEMS[5] := 0;
		Lynus_Standards.GVL_Energy.stDataElectricHeatingElements[diNrOfEMS_OUT,arrLPPrioZeroSetToZeroP[3]].arrTargetPowerEMS[6] := 0;
		Lynus_Standards.GVL_Energy.stDataElectricHeatingElements[diNrOfEMS_OUT,arrLPPrioZeroSetToZeroP[3]].arrTargetPowerEMS[7] := 0;
		Lynus_Standards.GVL_Energy.stDataElectricHeatingElements[diNrOfEMS_OUT,arrLPPrioZeroSetToZeroP[3]].arrTargetPowerEMS[8] := 0;
		Lynus_Standards.GVL_Energy.stDataElectricHeatingElements[diNrOfEMS_OUT,arrLPPrioZeroSetToZeroP[3]].arrTargetPowerEMS[9] := 0;
		Lynus_Standards.GVL_Energy.stDataElectricHeatingElements[diNrOfEMS_OUT,arrLPPrioZeroSetToZeroP[3]].arrTargetPowerEMS[10] := 0;
	END_IF
END_FOR
//OBC
FOR arrLPPrioZeroSetToZeroP[4] := 1 TO Constants_Energy.diMaxNumberOfOtherBigConsumers BY 1 DO
	IF Lynus_Standards.GVL_Energy.stDataOtherBigConsumers[diNrOfEMS_OUT,arrLPPrioZeroSetToZeroP[4]].byPriority = 0 OR Lynus_Standards.GVL_Energy.stDataOtherBigConsumers[diNrOfEMS_OUT,arrLPPrioZeroSetToZeroP[4]].byPriority > arrActualPrioInTurn[4] OR arrMinPrioReached[4] OR NOT bEnable OR FPEPO.Q OR 
	FNEPO.Q OR diMemCmpOperationState <> 0 OR eOperationMode = E_OperatingMode_EMS.eAllOff OR bStopAll THEN
		Lynus_Standards.GVL_Energy.stDataOtherBigConsumers[diNrOfEMS_OUT,arrLPPrioZeroSetToZeroP[4]].rTargetPowerEMS := 0;
	END_IF
END_FOR
//ECS
FOR arrLPPrioZeroSetToZeroP[5] := 1 TO Constants_Energy.diMaxNumberOfElectricChargingStations BY 1 DO
	IF Lynus_Standards.GVL_Energy.stDataElectricChargingStations[diNrOfEMS_OUT,arrLPPrioZeroSetToZeroP[5]].byPriority = 0 OR Lynus_Standards.GVL_Energy.stDataElectricChargingStations[diNrOfEMS_OUT,arrLPPrioZeroSetToZeroP[5]].byPriority > arrActualPrioInTurn[5] OR arrMinPrioReached[5] OR NOT bEnable OR FPEPO.Q OR FNEPO.Q OR 
	diMemCmpOperationState <> 0 OR eOperationMode = E_OperatingMode_EMS.eAllOff OR bStopAll OR 
	((eOperationMode = E_OperatingMode_EMS.ePeakLoadCapping OR eOperationMode = E_OperatingMode_EMS.eLoadManagement) AND stSetupEMS.bEnableMainFuseFunction AND (NOT Lynus_Standards.GVL_Energy.stDataElectricMeters[diNrOfEM_IN_ECS].bEnabled OR stSetupEMS.rSizeMainFuseCS <= 0 OR bDisableECS)) THEN
		Lynus_Standards.GVL_Energy.stDataElectricChargingStations[diNrOfEMS_OUT,arrLPPrioZeroSetToZeroP[5]].rTargetPowerEMS := 0;
	END_IF
END_FOR

(*----------------------------------------------------------------------------------------------------Controller to discharge/charge the batterys on the different modes----------------------------------------------------------------------------------------------------------*)
(*----------------------------------------------------------------------------------------------------Controller to discharge the battery in the self consumption mode----------------------------------------------------------------------------------------------------------*)

lrErrorPIDCorrectionBattSC := ABS(0 - lrGridPower);

//Controller weighting
IF eSpeedModeLocalController = E_SpeedModeLocalController_EMS.eSlow THEN 
	IF lrErrorPIDCorrectionBattSC <= 0.5 THEN 
		fbPIDBatterySC.rPValue := 0.05; fbPIDBatterySC.udiIValue := 450;
	ELSIF lrErrorPIDCorrectionBattSC > 0.5 AND lrErrorPIDCorrectionBattSC <= 1 THEN 
		fbPIDBatterySC.rPValue := 0.07; fbPIDBatterySC.udiIValue := 450;
	ELSIF lrErrorPIDCorrectionBattSC > 1 AND lrErrorPIDCorrectionBattSC <= 1.5 THEN 
		fbPIDBatterySC.rPValue := 0.09; fbPIDBatterySC.udiIValue := 450; 
	ELSIF lrErrorPIDCorrectionBattSC > 1.5 AND lrErrorPIDCorrectionBattSC <= 2 THEN 
		fbPIDBatterySC.rPValue := 0.11; fbPIDBatterySC.udiIValue := 450; 	
	ELSIF lrErrorPIDCorrectionBattSC > 2 AND lrErrorPIDCorrectionBattSC <= 2.5 THEN
		fbPIDBatterySC.rPValue := 0.13; fbPIDBatterySC.udiIValue := 675; 
	ELSIF lrErrorPIDCorrectionBattSC > 2.5 AND lrErrorPIDCorrectionBattSC <= 3 THEN
		fbPIDBatterySC.rPValue := 0.15; fbPIDBatterySC.udiIValue := 675;
	ELSIF lrErrorPIDCorrectionBattSC > 3 AND lrErrorPIDCorrectionBattSC <= 3.5 THEN 
		fbPIDBatterySC.rPValue := 0.17; fbPIDBatterySC.udiIValue := 900;
	ELSIF lrErrorPIDCorrectionBattSC > 3.5 AND lrErrorPIDCorrectionBattSC <= 4 THEN 
		fbPIDBatterySC.rPValue := 0.19; fbPIDBatterySC.udiIValue := 900;
	ELSIF lrErrorPIDCorrectionBattSC > 4 AND lrErrorPIDCorrectionBattSC <= 4.5 THEN 
		fbPIDBatterySC.rPValue := 0.21; fbPIDBatterySC.udiIValue := 900;
	ELSIF lrErrorPIDCorrectionBattSC > 4.5 AND lrErrorPIDCorrectionBattSC <= 5 THEN 
		fbPIDBatterySC.rPValue := 0.23; fbPIDBatterySC.udiIValue := 900;
	ELSIF lrErrorPIDCorrectionBattSC > 5 THEN 
		fbPIDBatterySC.rPValue := 0.25; fbPIDBatterySC.udiIValue := 900;
	END_IF
ELSIF eSpeedModeLocalController = E_SpeedModeLocalController_EMS.eBalanced THEN 
	IF lrErrorPIDCorrectionBattSC <= 0.5 THEN 
		fbPIDBatterySC.rPValue := 0.10; fbPIDBatterySC.udiIValue := 450;
	ELSIF lrErrorPIDCorrectionBattSC > 0.5 AND lrErrorPIDCorrectionBattSC <= 1 THEN 
		fbPIDBatterySC.rPValue := 0.14; fbPIDBatterySC.udiIValue := 450;
	ELSIF lrErrorPIDCorrectionBattSC > 1 AND lrErrorPIDCorrectionBattSC <= 1.5 THEN 
		fbPIDBatterySC.rPValue := 0.18; fbPIDBatterySC.udiIValue := 450; 
	ELSIF lrErrorPIDCorrectionBattSC > 1.5 AND lrErrorPIDCorrectionBattSC <= 2 THEN 
		fbPIDBatterySC.rPValue := 0.22; fbPIDBatterySC.udiIValue := 450; 	
	ELSIF lrErrorPIDCorrectionBattSC > 2 AND lrErrorPIDCorrectionBattSC <= 2.5 THEN 
		fbPIDBatterySC.rPValue := 0.26; fbPIDBatterySC.udiIValue := 675; 
	ELSIF lrErrorPIDCorrectionBattSC > 2.5 AND lrErrorPIDCorrectionBattSC <= 3 THEN 
		fbPIDBatterySC.rPValue := 0.30; fbPIDBatterySC.udiIValue := 675;
	ELSIF lrErrorPIDCorrectionBattSC > 3 AND lrErrorPIDCorrectionBattSC <= 3.5 THEN 
		fbPIDBatterySC.rPValue := 0.34; fbPIDBatterySC.udiIValue := 900;
	ELSIF lrErrorPIDCorrectionBattSC > 3.5 AND lrErrorPIDCorrectionBattSC <= 4 THEN 
		fbPIDBatterySC.rPValue := 0.38; fbPIDBatterySC.udiIValue := 900;
	ELSIF lrErrorPIDCorrectionBattSC > 4 AND lrErrorPIDCorrectionBattSC <= 4.5 THEN 
		fbPIDBatterySC.rPValue := 0.42; fbPIDBatterySC.udiIValue := 900;
	ELSIF lrErrorPIDCorrectionBattSC > 4.5 AND lrErrorPIDCorrectionBattSC <= 5 THEN 
		fbPIDBatterySC.rPValue := 0.46; fbPIDBatterySC.udiIValue := 900;
	ELSIF lrErrorPIDCorrectionBattSC > 5 THEN 
		fbPIDBatterySC.rPValue := 0.50; fbPIDBatterySC.udiIValue := 900;
	END_IF
ELSIF eSpeedModeLocalController = E_SpeedModeLocalController_EMS.eFast THEN
	IF lrErrorPIDCorrectionBattSC <= 0.5 THEN 
		fbPIDBatterySC.rPValue := 0.30; fbPIDBatterySC.udiIValue := 275;
	ELSIF lrErrorPIDCorrectionBattSC > 0.5 AND lrErrorPIDCorrectionBattSC <= 1 THEN 
		fbPIDBatterySC.rPValue := 0.33; fbPIDBatterySC.udiIValue := 275;
	ELSIF lrErrorPIDCorrectionBattSC > 1 AND lrErrorPIDCorrectionBattSC <= 1.5 THEN 
		fbPIDBatterySC.rPValue := 0.36; fbPIDBatterySC.udiIValue := 275; 
	ELSIF lrErrorPIDCorrectionBattSC > 1.5 AND lrErrorPIDCorrectionBattSC <= 2 THEN 
		fbPIDBatterySC.rPValue := 0.39; fbPIDBatterySC.udiIValue := 275; 	
	ELSIF lrErrorPIDCorrectionBattSC > 2 AND lrErrorPIDCorrectionBattSC <= 2.5 THEN 
		fbPIDBatterySC.rPValue := 0.42; fbPIDBatterySC.udiIValue := 500; 
	ELSIF lrErrorPIDCorrectionBattSC > 2.5 AND lrErrorPIDCorrectionBattSC <= 3 THEN 
		fbPIDBatterySC.rPValue := 0.45; fbPIDBatterySC.udiIValue := 500;
	ELSIF lrErrorPIDCorrectionBattSC > 3 AND lrErrorPIDCorrectionBattSC <= 3.5 THEN 
		fbPIDBatterySC.rPValue := 0.48; fbPIDBatterySC.udiIValue := 750;
	ELSIF lrErrorPIDCorrectionBattSC > 3.5 AND lrErrorPIDCorrectionBattSC <= 4 THEN 
		fbPIDBatterySC.rPValue := 0.51; fbPIDBatterySC.udiIValue := 750;
	ELSIF lrErrorPIDCorrectionBattSC > 4 AND lrErrorPIDCorrectionBattSC <= 4.5 THEN 
		fbPIDBatterySC.rPValue := 0.54; fbPIDBatterySC.udiIValue := 750;
	ELSIF lrErrorPIDCorrectionBattSC > 4.5 AND lrErrorPIDCorrectionBattSC <= 5 THEN 
		fbPIDBatterySC.rPValue := 0.57; fbPIDBatterySC.udiIValue := 750;
	ELSIF lrErrorPIDCorrectionBattSC > 5 THEN 
		fbPIDBatterySC.rPValue := 0.60; fbPIDBatterySC.udiIValue := 750;
	END_IF
END_IF

IF bEnable AND eOperationMode = E_OperatingMode_EMS.eSelfConsumption AND NOT bEPMActive AND NOT bStopAll AND NOT bDischrgCmdFromBackendOK AND 
arrMinPrioReached[1] AND arrMinPrioReached[2] AND arrMinPrioReached[3] AND arrMinPrioReached[4] AND arrMinPrioReached[5] THEN
	fbPIDBatterySC.bEnable := TRUE;
ELSE
	fbPIDBatterySC.bEnable := FALSE;
END_IF

fbPIDBatterySC( 
	bEnable:= , 
	rSetpoint:= 0, 
	udiIValue:= , 
	udiDValue:= 0, 
	udiDamping:= 0, 
	rPValue:= , 
	rMaxValue:= 100, 
	rMinValue:= 0, 
	rNeutralZone:= 0.1, 
	bDirection:= TRUE, 
	rActualValue:= LREAL_TO_REAL(lrGridPower), 
	rQController=> rControllerQPIDSC);

//Set the Controller output	to 0 when we have surplus. (Because its possible that the controller output is not set 100% to 0 regarding internal discrepancies)
IF rControllerQPIDSC <= 0.4 AND fbPIDBatterySC.bEnable AND lrGridPower <= - Constants_Energy.rToleranceSurplusConsumption THEN 
	timPIDSC.IN := TRUE;
ELSE
	timPIDSC.IN := FALSE;
END_IF

timPIDSC(IN:= , PT:= T#15S, Q=> , ET=> );
IF timPIDSC.Q THEN 
	rControllerQPIDSC := 0; 
END_IF	

FOR liLPDataBatteryInverter := 1 TO Constants_Energy.diMaxNumberOfBatteryInverters BY 1 DO
	IF Lynus_Standards.GVL_Energy.stDataOfBatteryInverters[diNrOfEMS_OUT,liLPDataBatteryInverter].byPriority <> 0 AND NOT bEPMActive AND eOperationMode = E_OperatingMode_EMS.eSelfConsumption AND	
	arrMinPrioReached[1] AND arrMinPrioReached[2] AND arrMinPrioReached[3] AND arrMinPrioReached[4] AND arrMinPrioReached[5] THEN
		Lynus_Standards.GVL_Energy.stDataOfBatteryInverters[diNrOfEMS_OUT,liLPDataBatteryInverter].rTargetPowerEMS := rControllerQPIDSC;
	END_IF 
END_FOR	

(*----------------------------------------------------------------------------------------------------Controller to charge and discharge the battery in the peak load capping mode and load management mode----------------------------------------------------------------------------------------------------------*)

//IMPORTANT : On this 2 modes the Batterys are allways active.
//This means that in these two modes the battery is not processed via the state machine like other devices.
//They are there to limit the power to the grid connection. The batteries charge according to the release when the power on the grid is below the grid connection or when power is fed back to the grid.
//The 95% are used so that the remaining 5% are still seen as surplus and thus the remaining consumers can still be regulated up to take advantage of the full grid connection.
//The batteries are processed with their priorities during charging. THIS means that only those batteries are active which also match the current active priority in the EMS.

(*--------------------------------------------------------------------------------------------------------------------Discharge the batterys-----------------------------------------------------------------------------------------------------------------------------------------------*)

lrErrorPIDCorrectionBattPLCLM_Dischrg := ABS(lrGridPower - (lrSizeGridConnection * 0.95));

//Controller weighting
IF eSpeedModeLocalController = E_SpeedModeLocalController_EMS.eSlow THEN 
	IF lrErrorPIDCorrectionBattPLCLM_Dischrg <= 0.5 THEN 
		fbPIDBatteryPLCLM_Dischrg.rPValue := 0.05; fbPIDBatteryPLCLM_Dischrg.udiIValue := 450;
	ELSIF lrErrorPIDCorrectionBattPLCLM_Dischrg > 0.5 AND lrErrorPIDCorrectionBattPLCLM_Dischrg <= 1 THEN 
		fbPIDBatteryPLCLM_Dischrg.rPValue := 0.07; fbPIDBatteryPLCLM_Dischrg.udiIValue := 450;
	ELSIF lrErrorPIDCorrectionBattPLCLM_Dischrg > 1 AND lrErrorPIDCorrectionBattPLCLM_Dischrg <= 1.5 THEN 
		fbPIDBatteryPLCLM_Dischrg.rPValue := 0.09; fbPIDBatteryPLCLM_Dischrg.udiIValue := 450; 
	ELSIF lrErrorPIDCorrectionBattPLCLM_Dischrg > 1.5 AND lrErrorPIDCorrectionBattPLCLM_Dischrg <= 2 THEN 
		fbPIDBatteryPLCLM_Dischrg.rPValue := 0.11; fbPIDBatteryPLCLM_Dischrg.udiIValue := 450; 	
	ELSIF lrErrorPIDCorrectionBattPLCLM_Dischrg > 2 AND lrErrorPIDCorrectionBattPLCLM_Dischrg <= 2.5 THEN 
		fbPIDBatteryPLCLM_Dischrg.rPValue := 0.13; fbPIDBatteryPLCLM_Dischrg.udiIValue := 675; 
	ELSIF lrErrorPIDCorrectionBattPLCLM_Dischrg > 2.5 AND lrErrorPIDCorrectionBattPLCLM_Dischrg <= 3 THEN 
		fbPIDBatteryPLCLM_Dischrg.rPValue := 0.15; fbPIDBatteryPLCLM_Dischrg.udiIValue := 675;
	ELSIF lrErrorPIDCorrectionBattPLCLM_Dischrg > 3 AND lrErrorPIDCorrectionBattPLCLM_Dischrg <= 3.5 THEN 
		fbPIDBatteryPLCLM_Dischrg.rPValue := 0.17; fbPIDBatteryPLCLM_Dischrg.udiIValue := 900;
	ELSIF lrErrorPIDCorrectionBattPLCLM_Dischrg > 3.5 AND lrErrorPIDCorrectionBattPLCLM_Dischrg <= 4 THEN 
		fbPIDBatteryPLCLM_Dischrg.rPValue := 0.19; fbPIDBatteryPLCLM_Dischrg.udiIValue := 900;
	ELSIF lrErrorPIDCorrectionBattPLCLM_Dischrg > 4 AND lrErrorPIDCorrectionBattPLCLM_Dischrg <= 4.5 THEN
		fbPIDBatteryPLCLM_Dischrg.rPValue := 0.21; fbPIDBatteryPLCLM_Dischrg.udiIValue := 900;
	ELSIF lrErrorPIDCorrectionBattPLCLM_Dischrg > 4.5 AND lrErrorPIDCorrectionBattPLCLM_Dischrg <= 5 THEN 
		fbPIDBatteryPLCLM_Dischrg.rPValue := 0.23; fbPIDBatteryPLCLM_Dischrg.udiIValue := 900;
	ELSIF lrErrorPIDCorrectionBattPLCLM_Dischrg > 5 THEN 
		fbPIDBatteryPLCLM_Dischrg.rPValue := 0.25; fbPIDBatteryPLCLM_Dischrg.udiIValue := 900;
	END_IF
ELSIF eSpeedModeLocalController = E_SpeedModeLocalController_EMS.eBalanced THEN
	IF lrErrorPIDCorrectionBattPLCLM_Dischrg <= 0.5 THEN 
		fbPIDBatteryPLCLM_Dischrg.rPValue := 0.10; fbPIDBatteryPLCLM_Dischrg.udiIValue := 450;
	ELSIF lrErrorPIDCorrectionBattPLCLM_Dischrg > 0.5 AND lrErrorPIDCorrectionBattPLCLM_Dischrg <= 1 THEN 
		fbPIDBatteryPLCLM_Dischrg.rPValue := 0.14; fbPIDBatteryPLCLM_Dischrg.udiIValue := 450;
	ELSIF lrErrorPIDCorrectionBattPLCLM_Dischrg > 1 AND lrErrorPIDCorrectionBattPLCLM_Dischrg <= 1.5 THEN 
		fbPIDBatteryPLCLM_Dischrg.rPValue := 0.18; fbPIDBatteryPLCLM_Dischrg.udiIValue := 450; 
	ELSIF lrErrorPIDCorrectionBattPLCLM_Dischrg > 1.5 AND lrErrorPIDCorrectionBattPLCLM_Dischrg <= 2 THEN 
		fbPIDBatteryPLCLM_Dischrg.rPValue := 0.22; fbPIDBatteryPLCLM_Dischrg.udiIValue := 450; 	
	ELSIF lrErrorPIDCorrectionBattPLCLM_Dischrg > 2 AND lrErrorPIDCorrectionBattPLCLM_Dischrg <= 2.5 THEN 
		fbPIDBatteryPLCLM_Dischrg.rPValue := 0.26; fbPIDBatteryPLCLM_Dischrg.udiIValue := 675; 
	ELSIF lrErrorPIDCorrectionBattPLCLM_Dischrg > 2.5 AND lrErrorPIDCorrectionBattPLCLM_Dischrg <= 3 THEN 
		fbPIDBatteryPLCLM_Dischrg.rPValue := 0.30; fbPIDBatteryPLCLM_Dischrg.udiIValue := 675;
	ELSIF lrErrorPIDCorrectionBattPLCLM_Dischrg > 3 AND lrErrorPIDCorrectionBattPLCLM_Dischrg <= 3.5 THEN 
		fbPIDBatteryPLCLM_Dischrg.rPValue := 0.34; fbPIDBatteryPLCLM_Dischrg.udiIValue := 900;
	ELSIF lrErrorPIDCorrectionBattPLCLM_Dischrg > 3.5 AND lrErrorPIDCorrectionBattPLCLM_Dischrg <= 4 THEN
		fbPIDBatteryPLCLM_Dischrg.rPValue := 0.38; fbPIDBatteryPLCLM_Dischrg.udiIValue := 900;
	ELSIF lrErrorPIDCorrectionBattPLCLM_Dischrg > 4 AND lrErrorPIDCorrectionBattPLCLM_Dischrg <= 4.5 THEN 
		fbPIDBatteryPLCLM_Dischrg.rPValue := 0.42; fbPIDBatteryPLCLM_Dischrg.udiIValue := 900;
	ELSIF lrErrorPIDCorrectionBattPLCLM_Dischrg > 4.5 AND lrErrorPIDCorrectionBattPLCLM_Dischrg <= 5 THEN 
		fbPIDBatteryPLCLM_Dischrg.rPValue := 0.46; fbPIDBatteryPLCLM_Dischrg.udiIValue := 900;
	ELSIF lrErrorPIDCorrectionBattPLCLM_Dischrg > 5 THEN 
		fbPIDBatteryPLCLM_Dischrg.rPValue := 0.50; fbPIDBatteryPLCLM_Dischrg.udiIValue := 900;
	END_IF
ELSIF eSpeedModeLocalController = E_SpeedModeLocalController_EMS.eFast THEN
	IF lrErrorPIDCorrectionBattPLCLM_Dischrg <= 0.5 THEN fbPIDBatteryPLCLM_Dischrg.rPValue := 0.30; fbPIDBatteryPLCLM_Dischrg.udiIValue := 275;
	ELSIF lrErrorPIDCorrectionBattPLCLM_Dischrg > 0.5 AND lrErrorPIDCorrectionBattPLCLM_Dischrg <= 1 THEN 
		fbPIDBatteryPLCLM_Dischrg.rPValue := 0.33; fbPIDBatteryPLCLM_Dischrg.udiIValue := 275;
	ELSIF lrErrorPIDCorrectionBattPLCLM_Dischrg > 1 AND lrErrorPIDCorrectionBattPLCLM_Dischrg <= 1.5 THEN 
		fbPIDBatteryPLCLM_Dischrg.rPValue := 0.36; fbPIDBatteryPLCLM_Dischrg.udiIValue := 275; 
	ELSIF lrErrorPIDCorrectionBattPLCLM_Dischrg > 1.5 AND lrErrorPIDCorrectionBattPLCLM_Dischrg <= 2 THEN 
		fbPIDBatteryPLCLM_Dischrg.rPValue := 0.39; fbPIDBatteryPLCLM_Dischrg.udiIValue := 275; 	
	ELSIF lrErrorPIDCorrectionBattPLCLM_Dischrg > 2 AND lrErrorPIDCorrectionBattPLCLM_Dischrg <= 2.5 THEN 
		fbPIDBatteryPLCLM_Dischrg.rPValue := 0.42; fbPIDBatteryPLCLM_Dischrg.udiIValue := 500; 
	ELSIF lrErrorPIDCorrectionBattPLCLM_Dischrg > 2.5 AND lrErrorPIDCorrectionBattPLCLM_Dischrg <= 3 THEN 
		fbPIDBatteryPLCLM_Dischrg.rPValue := 0.45; fbPIDBatteryPLCLM_Dischrg.udiIValue := 500;
	ELSIF lrErrorPIDCorrectionBattPLCLM_Dischrg > 3 AND lrErrorPIDCorrectionBattPLCLM_Dischrg <= 3.5 THEN 
		fbPIDBatteryPLCLM_Dischrg.rPValue := 0.48; fbPIDBatteryPLCLM_Dischrg.udiIValue := 750;
	ELSIF lrErrorPIDCorrectionBattPLCLM_Dischrg > 3.5 AND lrErrorPIDCorrectionBattPLCLM_Dischrg <= 4 THEN 
		fbPIDBatteryPLCLM_Dischrg.rPValue := 0.51; fbPIDBatteryPLCLM_Dischrg.udiIValue := 750;
	ELSIF lrErrorPIDCorrectionBattPLCLM_Dischrg > 4 AND lrErrorPIDCorrectionBattPLCLM_Dischrg <= 4.5 THEN 
		fbPIDBatteryPLCLM_Dischrg.rPValue := 0.54; fbPIDBatteryPLCLM_Dischrg.udiIValue := 750;
	ELSIF lrErrorPIDCorrectionBattPLCLM_Dischrg > 4.5 AND lrErrorPIDCorrectionBattPLCLM_Dischrg <= 5 THEN 
		fbPIDBatteryPLCLM_Dischrg.rPValue := 0.57; fbPIDBatteryPLCLM_Dischrg.udiIValue := 750;
	ELSIF lrErrorPIDCorrectionBattPLCLM_Dischrg > 5 THEN 
		fbPIDBatteryPLCLM_Dischrg.rPValue := 0.60; fbPIDBatteryPLCLM_Dischrg.udiIValue := 750;
	END_IF
END_IF 

IF (bEnable AND eOperationMode = E_OperatingMode_EMS.ePeakLoadCapping AND NOT bEPMActive AND NOT bStopAll AND NOT bDischrgCmdFromBackendOK AND NOT fbPIDBatteryPLCLM_Chrg.bEnable AND lrGridPower >= (lrSizeGridConnection * 0.95)) OR 
(bEnable AND eOperationMode = E_OperatingMode_EMS.eLoadManagement AND NOT bEPMActive AND NOT bStopAll AND NOT bDischrgCmdFromBackendOK AND NOT fbPIDBatteryPLCLM_Chrg.bEnable AND lrGridPower >= (SEL(bZeroPowerRegulation,lrSizeGridConnection,0) * 0.95)) THEN
	fbPIDBatteryPLCLM_Dischrg.bEnable := TRUE;
END_IF
IF NOT bEnable OR diNumberOfActiveBatterys = 0 OR bEPMActive OR bStopAll OR bDischrgCmdFromBackendOK OR fbPIDBatteryPLCLM_Chrg.bEnable OR eOperationMode = E_OperatingMode_EMS.eAllOff OR eOperationMode = E_OperatingMode_EMS.eSelfConsumption OR
(lrGridPower <SEL(bZeroPowerRegulation,(lrSizeGridConnection * 0.95),0) AND fbPIDBatteryPLCLM_Dischrg.rQController <= 0) THEN
	fbPIDBatteryPLCLM_Dischrg.bEnable := FALSE;
END_IF    

fbPIDBatteryPLCLM_Dischrg( 
	bEnable:= , 
	rSetpoint:=SEL(bZeroPowerRegulation,LREAL_TO_REAL(lrSizeGridConnection * 0.95),0), 
	udiIValue:= , 
	udiDValue:= 0, 
	udiDamping:= 0, 
	rPValue:= , 
	rMaxValue:= 100, 
	rMinValue:= 0, 
	rNeutralZone:= 0.1, 
	bDirection:= TRUE, 
	rActualValue:= LREAL_TO_REAL(lrGridPower), 
	rQController=> );

FOR liLPDataBatteryInverter := 1 TO Constants_Energy.diMaxNumberOfBatteryInverters BY 1 DO
	IF Lynus_Standards.GVL_Energy.stDataOfBatteryInverters[diNrOfEMS_OUT,liLPDataBatteryInverter].byPriority <> 0 AND NOT bEPMActive AND fbPIDBatteryPLCLM_Dischrg.bEnable THEN
		Lynus_Standards.GVL_Energy.stDataOfBatteryInverters[diNrOfEMS_OUT,liLPDataBatteryInverter].rTargetPowerEMS := fbPIDBatteryPLCLM_Dischrg.rQController;
	END_IF 
END_FOR	

(*--------------------------------------------------------------------------------------------------------------------Charge the batterys-----------------------------------------------------------------------------------------------------------------------------------------------*)

IF stSetupEMS.bAllowChrgFromGrid THEN 
	lrErrorPIDCorrectionBattPLCLM_Chrg := ABS(lrGridPower - (lrSizeGridConnection * 0.95));
ELSE
	lrErrorPIDCorrectionBattPLCLM_Chrg := ABS(0 - lrGridPower);
END_IF 

//Controller weighting
IF eSpeedModeLocalController = E_SpeedModeLocalController_EMS.eSlow THEN 
	IF lrErrorPIDCorrectionBattPLCLM_Chrg <= 0.5 THEN 
		fbPIDBatteryPLCLM_Chrg.rPValue := 0.05; fbPIDBatteryPLCLM_Chrg.udiIValue := 450;
	ELSIF lrErrorPIDCorrectionBattPLCLM_Chrg > 0.5 AND lrErrorPIDCorrectionBattPLCLM_Chrg <= 1 THEN 
		fbPIDBatteryPLCLM_Chrg.rPValue := 0.07; fbPIDBatteryPLCLM_Chrg.udiIValue := 450;
	ELSIF lrErrorPIDCorrectionBattPLCLM_Chrg > 1 AND lrErrorPIDCorrectionBattPLCLM_Chrg <= 1.5 THEN 
		fbPIDBatteryPLCLM_Chrg.rPValue := 0.09; fbPIDBatteryPLCLM_Chrg.udiIValue := 450; 
	ELSIF lrErrorPIDCorrectionBattPLCLM_Chrg > 1.5 AND lrErrorPIDCorrectionBattPLCLM_Chrg <= 2 THEN 
		fbPIDBatteryPLCLM_Chrg.rPValue := 0.11; fbPIDBatteryPLCLM_Chrg.udiIValue := 450; 	
	ELSIF lrErrorPIDCorrectionBattPLCLM_Chrg > 2 AND lrErrorPIDCorrectionBattPLCLM_Chrg <= 2.5 THEN 
		fbPIDBatteryPLCLM_Chrg.rPValue := 0.13; fbPIDBatteryPLCLM_Chrg.udiIValue := 675; 
	ELSIF lrErrorPIDCorrectionBattPLCLM_Chrg > 2.5 AND lrErrorPIDCorrectionBattPLCLM_Chrg <= 3 THEN 
		fbPIDBatteryPLCLM_Chrg.rPValue := 0.15; fbPIDBatteryPLCLM_Chrg.udiIValue := 675;
	ELSIF lrErrorPIDCorrectionBattPLCLM_Chrg > 3 AND lrErrorPIDCorrectionBattPLCLM_Chrg <= 3.5 THEN 
		fbPIDBatteryPLCLM_Chrg.rPValue := 0.17; fbPIDBatteryPLCLM_Chrg.udiIValue := 900;
	ELSIF lrErrorPIDCorrectionBattPLCLM_Chrg > 3.5 AND lrErrorPIDCorrectionBattPLCLM_Chrg <= 4 THEN 
		fbPIDBatteryPLCLM_Chrg.rPValue := 0.19; fbPIDBatteryPLCLM_Chrg.udiIValue := 900;
	ELSIF lrErrorPIDCorrectionBattPLCLM_Chrg > 4 AND lrErrorPIDCorrectionBattPLCLM_Chrg <= 4.5 THEN 
		fbPIDBatteryPLCLM_Chrg.rPValue := 0.21; fbPIDBatteryPLCLM_Chrg.udiIValue := 900;
	ELSIF lrErrorPIDCorrectionBattPLCLM_Chrg > 4.5 AND lrErrorPIDCorrectionBattPLCLM_Chrg <= 5 THEN 
		fbPIDBatteryPLCLM_Chrg.rPValue := 0.23; fbPIDBatteryPLCLM_Chrg.udiIValue := 900;
	ELSIF lrErrorPIDCorrectionBattPLCLM_Chrg > 5 THEN 
		fbPIDBatteryPLCLM_Chrg.rPValue := 0.25; fbPIDBatteryPLCLM_Chrg.udiIValue := 900;
	END_IF
ELSIF eSpeedModeLocalController = E_SpeedModeLocalController_EMS.eBalanced THEN
	IF lrErrorPIDCorrectionBattPLCLM_Chrg <= 0.5 THEN 
		fbPIDBatteryPLCLM_Chrg.rPValue := 0.10; fbPIDBatteryPLCLM_Chrg.udiIValue := 450;
	ELSIF lrErrorPIDCorrectionBattPLCLM_Chrg > 0.5 AND lrErrorPIDCorrectionBattPLCLM_Chrg <= 1 THEN 
		fbPIDBatteryPLCLM_Chrg.rPValue := 0.14; fbPIDBatteryPLCLM_Chrg.udiIValue := 450;
	ELSIF lrErrorPIDCorrectionBattPLCLM_Chrg > 1 AND lrErrorPIDCorrectionBattPLCLM_Chrg <= 1.5 THEN 
		fbPIDBatteryPLCLM_Chrg.rPValue := 0.18; fbPIDBatteryPLCLM_Chrg.udiIValue := 450; 
	ELSIF lrErrorPIDCorrectionBattPLCLM_Chrg > 1.5 AND lrErrorPIDCorrectionBattPLCLM_Chrg <= 2 THEN 
		fbPIDBatteryPLCLM_Chrg.rPValue := 0.22; fbPIDBatteryPLCLM_Chrg.udiIValue := 450; 	
	ELSIF lrErrorPIDCorrectionBattPLCLM_Chrg > 2 AND lrErrorPIDCorrectionBattPLCLM_Chrg <= 2.5 THEN 
		fbPIDBatteryPLCLM_Chrg.rPValue := 0.26; fbPIDBatteryPLCLM_Chrg.udiIValue := 675; 
	ELSIF lrErrorPIDCorrectionBattPLCLM_Chrg > 2.5 AND lrErrorPIDCorrectionBattPLCLM_Chrg <= 3 THEN 
		fbPIDBatteryPLCLM_Chrg.rPValue := 0.30; fbPIDBatteryPLCLM_Chrg.udiIValue := 675;
	ELSIF lrErrorPIDCorrectionBattPLCLM_Chrg > 3 AND lrErrorPIDCorrectionBattPLCLM_Chrg <= 3.5 THEN 
		fbPIDBatteryPLCLM_Chrg.rPValue := 0.34; fbPIDBatteryPLCLM_Chrg.udiIValue := 900;
	ELSIF lrErrorPIDCorrectionBattPLCLM_Chrg > 3.5 AND lrErrorPIDCorrectionBattPLCLM_Chrg <= 4 THEN 
		fbPIDBatteryPLCLM_Chrg.rPValue := 0.38; fbPIDBatteryPLCLM_Chrg.udiIValue := 900;
	ELSIF lrErrorPIDCorrectionBattPLCLM_Chrg > 4 AND lrErrorPIDCorrectionBattPLCLM_Chrg <= 4.5 THEN 
		fbPIDBatteryPLCLM_Chrg.rPValue := 0.42; fbPIDBatteryPLCLM_Chrg.udiIValue := 900;
	ELSIF lrErrorPIDCorrectionBattPLCLM_Chrg > 4.5 AND lrErrorPIDCorrectionBattPLCLM_Chrg <= 5 THEN 
		fbPIDBatteryPLCLM_Chrg.rPValue := 0.46; fbPIDBatteryPLCLM_Chrg.udiIValue := 900;
	ELSIF lrErrorPIDCorrectionBattPLCLM_Chrg > 5 THEN fbPIDBatteryPLCLM_Chrg.rPValue := 0.50; fbPIDBatteryPLCLM_Chrg.udiIValue := 900;
	END_IF
ELSIF eSpeedModeLocalController = E_SpeedModeLocalController_EMS.eFast THEN
	IF lrErrorPIDCorrectionBattPLCLM_Chrg <= 0.5 THEN 
		fbPIDBatteryPLCLM_Chrg.rPValue := 0.30; fbPIDBatteryPLCLM_Chrg.udiIValue := 275;
	ELSIF lrErrorPIDCorrectionBattPLCLM_Chrg > 0.5 AND lrErrorPIDCorrectionBattPLCLM_Chrg <= 1 THEN 
		fbPIDBatteryPLCLM_Chrg.rPValue := 0.33; fbPIDBatteryPLCLM_Chrg.udiIValue := 275;
	ELSIF lrErrorPIDCorrectionBattPLCLM_Chrg > 1 AND lrErrorPIDCorrectionBattPLCLM_Chrg <= 1.5 THEN 
		fbPIDBatteryPLCLM_Chrg.rPValue := 0.36; fbPIDBatteryPLCLM_Chrg.udiIValue := 275; 
	ELSIF lrErrorPIDCorrectionBattPLCLM_Chrg > 1.5 AND lrErrorPIDCorrectionBattPLCLM_Chrg <= 2 THEN 
		fbPIDBatteryPLCLM_Chrg.rPValue := 0.39; fbPIDBatteryPLCLM_Chrg.udiIValue := 275; 	
	ELSIF lrErrorPIDCorrectionBattPLCLM_Chrg > 2 AND lrErrorPIDCorrectionBattPLCLM_Chrg <= 2.5 THEN 
		fbPIDBatteryPLCLM_Chrg.rPValue := 0.42; fbPIDBatteryPLCLM_Chrg.udiIValue := 500; 
	ELSIF lrErrorPIDCorrectionBattPLCLM_Chrg > 2.5 AND lrErrorPIDCorrectionBattPLCLM_Chrg <= 3 THEN 
		fbPIDBatteryPLCLM_Chrg.rPValue := 0.45; fbPIDBatteryPLCLM_Chrg.udiIValue := 500;
	ELSIF lrErrorPIDCorrectionBattPLCLM_Chrg > 3 AND lrErrorPIDCorrectionBattPLCLM_Chrg <= 3.5 THEN 
		fbPIDBatteryPLCLM_Chrg.rPValue := 0.48; fbPIDBatteryPLCLM_Chrg.udiIValue := 750;
	ELSIF lrErrorPIDCorrectionBattPLCLM_Chrg > 3.5 AND lrErrorPIDCorrectionBattPLCLM_Chrg <= 4 THEN 
		fbPIDBatteryPLCLM_Chrg.rPValue := 0.51; fbPIDBatteryPLCLM_Chrg.udiIValue := 750;
	ELSIF lrErrorPIDCorrectionBattPLCLM_Chrg > 4 AND lrErrorPIDCorrectionBattPLCLM_Chrg <= 4.5 THEN 
		fbPIDBatteryPLCLM_Chrg.rPValue := 0.54; fbPIDBatteryPLCLM_Chrg.udiIValue := 750;
	ELSIF lrErrorPIDCorrectionBattPLCLM_Chrg > 4.5 AND lrErrorPIDCorrectionBattPLCLM_Chrg <= 5 THEN 
		fbPIDBatteryPLCLM_Chrg.rPValue := 0.57; fbPIDBatteryPLCLM_Chrg.udiIValue := 750;
	ELSIF lrErrorPIDCorrectionBattPLCLM_Chrg > 5 THEN 
		fbPIDBatteryPLCLM_Chrg.rPValue := 0.60; fbPIDBatteryPLCLM_Chrg.udiIValue := 750;
	END_IF	
END_IF

//Start and stop charge when charging from thr grid is allowed
IF (bEnable AND eOperationMode = E_OperatingMode_EMS.ePeakLoadCapping AND stSetupEMS.bAllowChrgFromGrid AND NOT bEPMActive AND NOT bStopAll AND NOT 
fbPIDBatteryPLCLM_Dischrg.bEnable AND NOT fbPIDDischrgCmdFromBackend.bEnable AND lrGridPower < (lrSizeGridConnection * 0.95)) AND (b_TimeBasedReleaseChargingBattery OR NOT b_EnableBatteryChargingControl) OR 
(bEnable AND eOperationMode = E_OperatingMode_EMS.eLoadManagement AND stSetupEMS.bAllowChrgFromGrid AND NOT bEPMActive AND NOT bStopAll AND NOT 
fbPIDBatteryPLCLM_Dischrg.bEnable AND NOT fbPIDDischrgCmdFromBackend.bEnable AND lrGridPower < (lrSizeGridConnection * 0.95)) THEN
	fbPIDBatteryPLCLM_Chrg.bEnable := TRUE;
END_IF
IF (stSetupEMS.bAllowChrgFromGrid AND (NOT bEnable OR diNumberOfActiveBatterys = 0 OR bEPMActive OR bStopAll OR fbPIDBatteryPLCLM_Dischrg.bEnable OR eOperationMode = E_OperatingMode_EMS.eAllOff OR 
eOperationMode = E_OperatingMode_EMS.eSelfConsumption OR fbPIDDischrgCmdFromBackend.bEnable OR (fbPIDBatteryPLCLM_Chrg.rQController >= 0 AND lrGridPower >= (lrSizeGridConnection * 0.95)))) OR NOT b_TimeBasedReleaseChargingBattery THEN
	fbPIDBatteryPLCLM_Chrg.bEnable := FALSE;
END_IF

//Start and stop charge when charging from thr grid is not allowed
IF (bEnable AND eOperationMode = E_OperatingMode_EMS.ePeakLoadCapping AND NOT stSetupEMS.bAllowChrgFromGrid AND NOT bEPMActive AND NOT bStopAll AND NOT 
fbPIDBatteryPLCLM_Dischrg.bEnable AND NOT fbPIDDischrgCmdFromBackend.bEnable AND lrGridPower < 0) OR 
(bEnable AND eOperationMode = E_OperatingMode_EMS.eLoadManagement AND NOT stSetupEMS.bAllowChrgFromGrid AND NOT bEPMActive AND NOT bStopAll AND NOT 
fbPIDBatteryPLCLM_Dischrg.bEnable AND NOT fbPIDDischrgCmdFromBackend.bEnable AND lrGridPower < 0) THEN
	fbPIDBatteryPLCLM_Chrg.bEnable := TRUE;
END_IF
IF (NOT stSetupEMS.bAllowChrgFromGrid AND (NOT bEnable OR diNumberOfActiveBatterys = 0 OR bEPMActive OR bStopAll OR fbPIDBatteryPLCLM_Dischrg.bEnable OR eOperationMode = E_OperatingMode_EMS.eAllOff OR 
eOperationMode = E_OperatingMode_EMS.eSelfConsumption OR fbPIDDischrgCmdFromBackend.bEnable OR (fbPIDBatteryPLCLM_Chrg.rQController >= 0 AND lrGridPower >= 0))) THEN
	fbPIDBatteryPLCLM_Chrg.bEnable := FALSE;
END_IF

//Set the Setpoint from the controller	
IF stSetupEMS.bAllowChrgFromGrid AND dwAvarageBatterySOC < stSetupEMS.byResChrgfromGridToBatt THEN 
	fbPIDBatteryPLCLM_Chrg.rSetpoint := LREAL_TO_REAL(lrSizeGridConnection * 0.95);
ELSE
	fbPIDBatteryPLCLM_Chrg.rSetpoint := 0;
END_IF 	
	
fbPIDBatteryPLCLM_Chrg( 
	bEnable:= , 
	rSetpoint:= , 
	udiIValue:= , 
	udiDValue:= 0, 
	udiDamping:= 0, 
	rPValue:= , 
	rMaxValue:= 0, 
	rMinValue:= rMaxBattChargingPower *(-1),
	rNeutralZone:= 0.1, 
	bDirection:= TRUE, 
	rActualValue:= LREAL_TO_REAL(lrGridPower), 
	rQController=> );

FOR liLPDataBatteryInverter := 1 TO Constants_Energy.diMaxNumberOfBatteryInverters BY 1 DO
	IF Lynus_Standards.GVL_Energy.stDataOfBatteryInverters[diNrOfEMS_OUT,liLPDataBatteryInverter].byPriority <= bySmGrActiveCommonPrio AND Lynus_Standards.GVL_Energy.stDataOfBatteryInverters[diNrOfEMS_OUT,liLPDataBatteryInverter].byPriority <> 0 AND NOT 
	bEPMActive AND fbPIDBatteryPLCLM_Chrg.bEnable THEN
		Lynus_Standards.GVL_Energy.stDataOfBatteryInverters[diNrOfEMS_OUT,liLPDataBatteryInverter].rTargetPowerEMS := fbPIDBatteryPLCLM_Chrg.rQController;
	END_IF 
END_FOR	

(*----------------------------------------------------------------------------------------------------Controller to discharge the battery in the emergency power mode----------------------------------------------------------------------------------------------------------*)

//All batterys what made active a island grid (Emergency power mode), the receive a target power form -100% to charge. The rest of the logic must implementet in each battery or batteryinverter function.
//Calculates the power from all batterys wich made a island grid
lrSizeBatteryPowerInEPO := 0;
FOR liLPDataBatteryInverter := 1 TO Constants_Energy.diMaxNumberOfBatteryInverters BY 1 DO
	IF Lynus_Standards.GVL_Energy.stDataOfBatteryInverters[diNrOfEMS_OUT,liLPDataBatteryInverter].bWorkOnIslandMode AND bEPMActive AND NOT bStopAll THEN 
		Lynus_Standards.GVL_Energy.stDataOfBatteryInverters[diNrOfEMS_OUT,liLPDataBatteryInverter].rTargetPowerEMS := -100; 
		lrSizeBatteryPowerInEPO := lrSizeBatteryPowerInEPO + Lynus_Standards.GVL_Energy.stDataOfBatteryInverters[diNrOfEMS_OUT,liLPDataBatteryInverter].lrPowerOnIslandMode;  
	END_IF
END_FOR	

lrErrorPIDCorrectionBattEPO := ABS(0 - lrSizeBatteryPowerInEPO);

//Controller weighting
IF eSpeedModeLocalController = E_SpeedModeLocalController_EMS.eSlow THEN
	IF lrErrorPIDCorrectionBattEPO <= 0.5 THEN 
		fbPIDBatteryEPO.rPValue := 0.05; fbPIDBatteryEPO.udiIValue := 450;
	ELSIF lrErrorPIDCorrectionBattEPO > 0.5 AND lrErrorPIDCorrectionBattEPO <= 1 THEN 
		fbPIDBatteryEPO.rPValue := 0.07; fbPIDBatteryEPO.udiIValue := 450;
	ELSIF lrErrorPIDCorrectionBattEPO > 1 AND lrErrorPIDCorrectionBattEPO <= 1.5 THEN 
		fbPIDBatteryEPO.rPValue := 0.09; fbPIDBatteryEPO.udiIValue := 450; 
	ELSIF lrErrorPIDCorrectionBattEPO > 1.5 AND lrErrorPIDCorrectionBattEPO <= 2 THEN 
		fbPIDBatteryEPO.rPValue := 0.11; fbPIDBatteryEPO.udiIValue := 450; 	
	ELSIF lrErrorPIDCorrectionBattEPO > 2 AND lrErrorPIDCorrectionBattEPO <= 2.5 THEN 
		fbPIDBatteryEPO.rPValue := 0.13; fbPIDBatteryEPO.udiIValue := 675; 
	ELSIF lrErrorPIDCorrectionBattEPO > 2.5 AND lrErrorPIDCorrectionBattEPO <= 3 THEN 
		fbPIDBatteryEPO.rPValue := 0.15; fbPIDBatteryEPO.udiIValue := 675;
	ELSIF lrErrorPIDCorrectionBattEPO > 3 AND lrErrorPIDCorrectionBattEPO <= 3.5 THEN 
		fbPIDBatteryEPO.rPValue := 0.17; fbPIDBatteryEPO.udiIValue := 900;
	ELSIF lrErrorPIDCorrectionBattEPO > 3.5 AND lrErrorPIDCorrectionBattEPO <= 4 THEN 
		fbPIDBatteryEPO.rPValue := 0.19; fbPIDBatteryEPO.udiIValue := 900;
	ELSIF lrErrorPIDCorrectionBattEPO > 4 AND lrErrorPIDCorrectionBattEPO <= 4.5 THEN 
		fbPIDBatteryEPO.rPValue := 0.21; fbPIDBatteryEPO.udiIValue := 900;
	ELSIF lrErrorPIDCorrectionBattEPO > 4.5 AND lrErrorPIDCorrectionBattEPO <= 5 THEN 
		fbPIDBatteryEPO.rPValue := 0.23; fbPIDBatteryEPO.udiIValue := 900;
	ELSIF lrErrorPIDCorrectionBattEPO > 5 THEN 
		fbPIDBatteryEPO.rPValue := 0.25; fbPIDBatteryEPO.udiIValue := 900;
	END_IF
ELSIF eSpeedModeLocalController = E_SpeedModeLocalController_EMS.eBalanced THEN
	IF lrErrorPIDCorrectionBattEPO <= 0.5 THEN 
		fbPIDBatteryEPO.rPValue := 0.10; fbPIDBatteryEPO.udiIValue := 450;
	ELSIF lrErrorPIDCorrectionBattEPO > 0.5 AND lrErrorPIDCorrectionBattEPO <= 1 THEN 
		fbPIDBatteryEPO.rPValue := 0.14; fbPIDBatteryEPO.udiIValue := 450;
	ELSIF lrErrorPIDCorrectionBattEPO > 1 AND lrErrorPIDCorrectionBattEPO <= 1.5 THEN 
		fbPIDBatteryEPO.rPValue := 0.18; fbPIDBatteryEPO.udiIValue := 450; 
	ELSIF lrErrorPIDCorrectionBattEPO > 1.5 AND lrErrorPIDCorrectionBattEPO <= 2 THEN 
		fbPIDBatteryEPO.rPValue := 0.22; fbPIDBatteryEPO.udiIValue := 450; 	
	ELSIF lrErrorPIDCorrectionBattEPO > 2 AND lrErrorPIDCorrectionBattEPO <= 2.5 THEN 
		fbPIDBatteryEPO.rPValue := 0.26; fbPIDBatteryEPO.udiIValue := 675; 
	ELSIF lrErrorPIDCorrectionBattEPO > 2.5 AND lrErrorPIDCorrectionBattEPO <= 3 THEN 
		fbPIDBatteryEPO.rPValue := 0.30; fbPIDBatteryEPO.udiIValue := 675;
	ELSIF lrErrorPIDCorrectionBattEPO > 3 AND lrErrorPIDCorrectionBattEPO <= 3.5 THEN 
		fbPIDBatteryEPO.rPValue := 0.34; fbPIDBatteryEPO.udiIValue := 900;
	ELSIF lrErrorPIDCorrectionBattEPO > 3.5 AND lrErrorPIDCorrectionBattEPO <= 4 THEN 
		fbPIDBatteryEPO.rPValue := 0.38; fbPIDBatteryEPO.udiIValue := 900;
	ELSIF lrErrorPIDCorrectionBattEPO > 4 AND lrErrorPIDCorrectionBattEPO <= 4.5 THEN 
		fbPIDBatteryEPO.rPValue := 0.42; fbPIDBatteryEPO.udiIValue := 900;
	ELSIF lrErrorPIDCorrectionBattEPO > 4.5 AND lrErrorPIDCorrectionBattEPO <= 5 THEN 
		fbPIDBatteryEPO.rPValue := 0.46; fbPIDBatteryEPO.udiIValue := 900;
	ELSIF lrErrorPIDCorrectionBattEPO > 5 THEN 
		fbPIDBatteryEPO.rPValue := 0.50; fbPIDBatteryEPO.udiIValue := 900;
	END_IF
ELSIF eSpeedModeLocalController = E_SpeedModeLocalController_EMS.eFast THEN
	IF lrErrorPIDCorrectionBattEPO <= 0.5 THEN 
		fbPIDBatteryEPO.rPValue := 0.30; fbPIDBatteryEPO.udiIValue := 275;
	ELSIF lrErrorPIDCorrectionBattEPO > 0.5 AND lrErrorPIDCorrectionBattEPO <= 1 THEN 
		fbPIDBatteryEPO.rPValue := 0.33; fbPIDBatteryEPO.udiIValue := 275;
	ELSIF lrErrorPIDCorrectionBattEPO > 1 AND lrErrorPIDCorrectionBattEPO <= 1.5 THEN 
		fbPIDBatteryEPO.rPValue := 0.36; fbPIDBatteryEPO.udiIValue := 275; 
	ELSIF lrErrorPIDCorrectionBattEPO > 1.5 AND lrErrorPIDCorrectionBattEPO <= 2 THEN 
		fbPIDBatteryEPO.rPValue := 0.39; fbPIDBatteryEPO.udiIValue := 275; 	
	ELSIF lrErrorPIDCorrectionBattEPO > 2 AND lrErrorPIDCorrectionBattEPO <= 2.5 THEN 
		fbPIDBatteryEPO.rPValue := 0.42; fbPIDBatteryEPO.udiIValue := 500; 
	ELSIF lrErrorPIDCorrectionBattEPO > 2.5 AND lrErrorPIDCorrectionBattEPO <= 3 THEN 
		fbPIDBatteryEPO.rPValue := 0.45; fbPIDBatteryEPO.udiIValue := 500;
	ELSIF lrErrorPIDCorrectionBattEPO > 3 AND lrErrorPIDCorrectionBattEPO <= 3.5 THEN 
		fbPIDBatteryEPO.rPValue := 0.48; fbPIDBatteryEPO.udiIValue := 750;
	ELSIF lrErrorPIDCorrectionBattEPO > 3.5 AND lrErrorPIDCorrectionBattEPO <= 4 THEN 
		fbPIDBatteryEPO.rPValue := 0.51; fbPIDBatteryEPO.udiIValue := 750;
	ELSIF lrErrorPIDCorrectionBattEPO > 4 AND lrErrorPIDCorrectionBattEPO <= 4.5 THEN 
		fbPIDBatteryEPO.rPValue := 0.54; fbPIDBatteryEPO.udiIValue := 750;
	ELSIF lrErrorPIDCorrectionBattEPO > 4.5 AND lrErrorPIDCorrectionBattEPO <= 5 THEN 
		fbPIDBatteryEPO.rPValue := 0.57; fbPIDBatteryEPO.udiIValue := 750;
	ELSIF lrErrorPIDCorrectionBattEPO > 5 THEN 
		fbPIDBatteryEPO.rPValue := 0.60; fbPIDBatteryEPO.udiIValue := 750;
	END_IF
END_IF

IF bEnable AND bEPMActive AND arrMinPrioReached[1] AND arrMinPrioReached[2] AND arrMinPrioReached[3] AND arrMinPrioReached[4] AND arrMinPrioReached[5] AND NOT bChargePrioBatterysOnEPO AND NOT bStopAll THEN
	fbPIDBatteryEPO.bEnable := TRUE;
ELSE
	fbPIDBatteryEPO.bEnable := FALSE;
END_IF

fbPIDBatteryEPO(
	bEnable:= , 
	rSetpoint:= 0, 
	udiIValue:= , 
	udiDValue:= 0, 
	udiDamping:= 0, 
	rPValue:= , 
	rMaxValue:= 100, 
	rMinValue:= 0, 
	rNeutralZone:= 0.1, 
	bDirection:= TRUE, 
	rActualValue:= LREAL_TO_REAL(lrSizeBatteryPowerInEPO), 
	rQController=> rControllerQPIDEPO);

//Set the Controller output	to 0 when we have surplus. (Because its possible that the controller output is not set 100% to 0 regarding internal discrepancies)
IF rControllerQPIDEPO <= 0.4 AND fbPIDBatteryEPO.bEnable AND lrSizeBatteryPowerInEPO <= - Constants_Energy.rToleranceSurplusConsumption THEN
	timPIDEPO.IN := TRUE;
ELSE
	timPIDEPO.IN := FALSE;
END_IF
	
timPIDEPO(IN:= , PT:= T#15S, Q=> , ET=> );
IF timPIDEPO.Q THEN 
	rControllerQPIDEPO := 0; 
END_IF

FOR liLPDataBatteryInverter := 1 TO Constants_Energy.diMaxNumberOfBatteryInverters BY 1 DO
	IF Lynus_Standards.GVL_Energy.stDataOfBatteryInverters[diNrOfEMS_OUT,liLPDataBatteryInverter].byPriority <> 0 AND bEPMActive AND NOT Lynus_Standards.GVL_Energy.stDataOfBatteryInverters[diNrOfEMS_OUT,liLPDataBatteryInverter].bWorkOnIslandMode AND 
	arrMinPrioReached[1] AND arrMinPrioReached[2] AND arrMinPrioReached[3] AND arrMinPrioReached[4] AND arrMinPrioReached[5] AND NOT bChargePrioBatterysOnEPO THEN
		Lynus_Standards.GVL_Energy.stDataOfBatteryInverters[diNrOfEMS_OUT,liLPDataBatteryInverter].rTargetPowerEMS := rControllerQPIDEPO;
	END_IF
END_FOR 

(*-----------------------------------------------------------Controll the Batterys and Heating pumps with the Backend Commands-----------------------------------------------------------------*)

//Controll the Heating Pumps
FOR liLPDischrgCmdFromBackend := 1 TO Constants_Energy.diMaxNumberOfHeatingPumps BY 1 DO  
	IF timErrorWarning.Q AND timEnergyOptReady.Q AND NOT timHB.Q THEN 
		Lynus_Standards.GVL_Energy.stDataHeatingPumps[diNrOfEMS_OUT,liLPDischrgCmdFromBackend].bExternalOnCommand := bActivateHP; 
	ELSE
		Lynus_Standards.GVL_Energy.stDataHeatingPumps[diNrOfEMS_OUT,liLPDischrgCmdFromBackend].bExternalOnCommand := FALSE;
	END_IF
END_FOR
//Reset the Activation from the HP (Maybe when we have communicaiton Error with the backend in this time when he well reset the command or somthing else...)
timResetActivateHP(IN:= bActivateHP, PT:= T#2M, Q=> , ET=> );
IF timResetActivateHP.Q THEN 
	bActivateHP := FALSE; 
END_IF

//Controll the discharge power from the Batterys with the power command from the Backend
//Calculate the actual Battery Power
lrActualPowerBatterys := 0;
FOR liLPDischrgCmdFromBackend := 1 TO Constants_Energy.diMaxNumberOfBatterys BY 1 DO
	lrActualPowerBatterys := lrActualPowerBatterys + Lynus_Standards.GVL_Energy.stDataOfBatterys[diNrOfEMS_OUT,liLPDischrgCmdFromBackend].lrPower;	
END_FOR

//Reset the Controller when we have surplus in the slef consumption mode
IF bSurplusAvailable AND eOperationMode = E_OperatingMode_EMS.eSelfConsumption THEN 
	timPIDDischrgCmdFromBackend.IN := TRUE;
ELSE
	timPIDDischrgCmdFromBackend.IN := FALSE;
END_IF

//Reset the Controller when we have surplus in the Load capping or load management mode
IF ((eOperationMode = E_OperatingMode_EMS.eLoadManagement OR eOperationMode = E_OperatingMode_EMS.ePeakLoadCapping) AND (lrGridPower < (lrSizeGridConnection * 0.95))) THEN
	timPIDDischrgCmdFromBackend.IN := TRUE;
END_IF
IF ((eOperationMode = E_OperatingMode_EMS.eLoadManagement OR eOperationMode = E_OperatingMode_EMS.ePeakLoadCapping) AND (lrGridPower >= (lrSizeGridConnection * 0.95))) THEN
	timPIDDischrgCmdFromBackend.IN := FALSE;
END_IF	  

//Give the Controller 35 Seconds Time. So he can make 3 times a correction for the power when the Backend commands to much Battery power.
timPIDDischrgCmdFromBackend(IN:= , PT:= T#35S, Q=> , ET=> );

//Enable or dissable the controller when Self Consumption mode is active
IF bEnable AND NOT bEPMActive AND NOT bStopAll AND bDischrgCmdFromBackendOK AND eOperationMode <> E_OperatingMode_EMS.eAllOff AND diMemCmpOperationState = 0 AND 
arrMinPrioReached[1] AND arrMinPrioReached[2] AND arrMinPrioReached[3] AND arrMinPrioReached[4] AND arrMinPrioReached[5] AND NOT timPIDDischrgCmdFromBackend.Q AND eOperationMode = E_OperatingMode_EMS.eSelfConsumption THEN
	fbPIDDischrgCmdFromBackend.bEnable := TRUE;
ELSE
	fbPIDDischrgCmdFromBackend.bEnable := FALSE;
END_IF	

//Enable or dissable the controller when Paeak Load capping or load management mode is active
IF bEnable AND NOT bEPMActive AND NOT bStopAll AND bDischrgCmdFromBackendOK AND eOperationMode <> E_OperatingMode_EMS.eAllOff AND diMemCmpOperationState = 0 AND 
eOperationMode = E_OperatingMode_EMS.eLoadManagement AND NOT fbPIDBatteryPLCLM_Chrg.bEnable AND NOT timPIDDischrgCmdFromBackend.Q THEN
	fbPIDDischrgCmdFromBackend.bEnable := TRUE;
END_IF	
IF eOperationMode = E_OperatingMode_EMS.eLoadManagement AND (NOT bEnable OR diNumberOfActiveBatterys = 0 OR bEPMActive OR bStopAll OR fbPIDBatteryPLCLM_Chrg.bEnable OR timPIDDischrgCmdFromBackend.Q) THEN 
	fbPIDDischrgCmdFromBackend.bEnable := FALSE; 
END_IF

IF bEnable AND NOT bEPMActive AND NOT bStopAll AND bDischrgCmdFromBackendOK AND eOperationMode <> E_OperatingMode_EMS.eAllOff AND diMemCmpOperationState = 0 AND 
eOperationMode = E_OperatingMode_EMS.ePeakLoadCapping AND NOT fbPIDBatteryPLCLM_Chrg.bEnable AND NOT timPIDDischrgCmdFromBackend.Q THEN
	fbPIDDischrgCmdFromBackend.bEnable := TRUE;
END_IF	
IF eOperationMode = E_OperatingMode_EMS.ePeakLoadCapping AND (NOT bEnable OR diNumberOfActiveBatterys = 0 OR bEPMActive OR bStopAll OR fbPIDBatteryPLCLM_Chrg.bEnable OR timPIDDischrgCmdFromBackend.Q) THEN 
	fbPIDDischrgCmdFromBackend.bEnable := FALSE; 
END_IF 

//Correction and safety for the Setpoint, that we dont give power back to the grid
//Set one time the new received Battery power and make then the correction (New reveived value from Backend or the PID Controller start from new)
FPEnablePID(CLK:= fbPIDDischrgCmdFromBackend.bEnable, Q=> );
IF rNewBattPower <> rNewBattPower_CP OR FPEnablePID.Q THEN
	lrNewBatteryPowerWithCorrection := rNewBattPower;
	rNewBattPower_CP := rNewBattPower;
END_IF

//Give the Controller and the Inverter time to set the new Setpoint
IF lrGridPower <> lrGridPower_CP AND NOT timCorrectionSetpoint.Q  AND bDischrgCmdFromBackendOK THEN
	timCorrectionSetpoint.IN := TRUE;
	lrGridPower_CP := lrGridPower;
ELSE
	timCorrectionSetpoint.IN := FALSE;
END_IF	 

//Make the correction a litte bit faster when the power on the grid is not so big
timCorrectionSetpoint.PT := T#10S;
IF lrGridPower >= - 0.30 AND lrGridPower <= 0.30 THEN 
	timCorrectionSetpoint.PT := T#7.5S; 
END_IF
IF lrGridPower >= - 0.20 AND lrGridPower <= 0.20 THEN 
	timCorrectionSetpoint.PT := T#5S; 
END_IF

timCorrectionSetpoint(IN:= , PT:= , Q=> , ET=> );
FPMakeCorrection(CLK:= timCorrectionSetpoint.Q, Q=> );

//Batterycorrection when Self Consumption Mode is active
IF FPMakeCorrection.Q AND eOperationMode = E_OperatingMode_EMS.eSelfConsumption THEN
	lrNewBatteryPowerWithCorrection := lrNewBatteryPowerWithCorrection + lrGridPower;
END_IF
//Batterycorrection when Peak load capping or load management Mode is active
IF FPMakeCorrection.Q AND eOperationMode = E_OperatingMode_EMS.eLoadManagement OR eOperationMode = E_OperatingMode_EMS.ePeakLoadCapping THEN
	lrNewBatteryPowerWithCorrection := (lrNewBatteryPowerWithCorrection + (lrGridPower - (lrSizeGridConnection * 0.96)));
END_IF

IF lrNewBatteryPowerWithCorrection < 0 THEN 
	lrNewBatteryPowerWithCorrection := 0; 
END_IF
IF lrNewBatteryPowerWithCorrection > rNewBattPower THEN 
	lrNewBatteryPowerWithCorrection := rNewBattPower; 
END_IF 

lrErrorPIDCorrectionDischrgCmdFromBackend := ABS(lrNewBatteryPowerWithCorrection - lrActualPowerBatterys);

//Controller weighting
IF eSpeedModeBackendController = E_SpeedModeBackendController_EMS.eSlow THEN
	IF lrErrorPIDCorrectionDischrgCmdFromBackend <= 0.5 THEN 
		fbPIDDischrgCmdFromBackend.rPValue := 0.05; 
		fbPIDDischrgCmdFromBackend.udiIValue := 450;
	ELSIF lrErrorPIDCorrectionDischrgCmdFromBackend > 0.5 AND lrErrorPIDCorrectionDischrgCmdFromBackend <= 1 THEN 
		fbPIDDischrgCmdFromBackend.rPValue := 0.07; 
		fbPIDDischrgCmdFromBackend.udiIValue := 450;
	ELSIF lrErrorPIDCorrectionDischrgCmdFromBackend > 1 AND lrErrorPIDCorrectionDischrgCmdFromBackend <= 1.5 THEN 
		fbPIDDischrgCmdFromBackend.rPValue := 0.09; 
		fbPIDDischrgCmdFromBackend.udiIValue := 450; 
	ELSIF lrErrorPIDCorrectionDischrgCmdFromBackend > 1.5 AND lrErrorPIDCorrectionDischrgCmdFromBackend <= 2 THEN 
		fbPIDDischrgCmdFromBackend.rPValue := 0.11; 
		fbPIDDischrgCmdFromBackend.udiIValue := 450; 	
	ELSIF lrErrorPIDCorrectionDischrgCmdFromBackend > 2 AND lrErrorPIDCorrectionDischrgCmdFromBackend <= 2.5 THEN 
		fbPIDDischrgCmdFromBackend.rPValue := 0.13; 
		fbPIDDischrgCmdFromBackend.udiIValue := 675; 
	ELSIF lrErrorPIDCorrectionDischrgCmdFromBackend > 2.5 AND lrErrorPIDCorrectionDischrgCmdFromBackend <= 3 THEN 
		fbPIDDischrgCmdFromBackend.rPValue := 0.15; 
		fbPIDDischrgCmdFromBackend.udiIValue := 675;
	ELSIF lrErrorPIDCorrectionDischrgCmdFromBackend > 3 AND lrErrorPIDCorrectionDischrgCmdFromBackend <= 3.5 THEN 
		fbPIDDischrgCmdFromBackend.rPValue := 0.17; 
		fbPIDDischrgCmdFromBackend.udiIValue := 900;
	ELSIF lrErrorPIDCorrectionDischrgCmdFromBackend > 3.5 AND lrErrorPIDCorrectionDischrgCmdFromBackend <= 4 THEN 
		fbPIDDischrgCmdFromBackend.rPValue := 0.19; 
		fbPIDDischrgCmdFromBackend.udiIValue := 900;
	ELSIF lrErrorPIDCorrectionDischrgCmdFromBackend > 4 AND lrErrorPIDCorrectionDischrgCmdFromBackend <= 4.5 THEN 
		fbPIDDischrgCmdFromBackend.rPValue := 0.21; 
		fbPIDDischrgCmdFromBackend.udiIValue := 900;
	ELSIF lrErrorPIDCorrectionDischrgCmdFromBackend > 4.5 AND lrErrorPIDCorrectionDischrgCmdFromBackend <= 5 THEN 
		fbPIDDischrgCmdFromBackend.rPValue := 0.23; 
		fbPIDDischrgCmdFromBackend.udiIValue := 900;
	ELSIF lrErrorPIDCorrectionDischrgCmdFromBackend > 5 THEN 
		fbPIDDischrgCmdFromBackend.rPValue := 0.25; 
		fbPIDDischrgCmdFromBackend.udiIValue := 900;
	END_IF
ELSIF eSpeedModeBackendController = E_SpeedModeBackendController_EMS.eBalanced THEN
	IF lrErrorPIDCorrectionDischrgCmdFromBackend <= 0.5 THEN 
		fbPIDDischrgCmdFromBackend.rPValue := 0.10; 
		fbPIDDischrgCmdFromBackend.udiIValue := 450;
	ELSIF lrErrorPIDCorrectionDischrgCmdFromBackend > 0.5 AND lrErrorPIDCorrectionDischrgCmdFromBackend <= 1 THEN 
		fbPIDDischrgCmdFromBackend.rPValue := 0.14; 
		fbPIDDischrgCmdFromBackend.udiIValue := 450;
	ELSIF lrErrorPIDCorrectionDischrgCmdFromBackend > 1 AND lrErrorPIDCorrectionDischrgCmdFromBackend <= 1.5 THEN 
		fbPIDDischrgCmdFromBackend.rPValue := 0.18; 
		fbPIDDischrgCmdFromBackend.udiIValue := 450; 
	ELSIF lrErrorPIDCorrectionDischrgCmdFromBackend > 1.5 AND lrErrorPIDCorrectionDischrgCmdFromBackend <= 2 THEN 
		fbPIDDischrgCmdFromBackend.rPValue := 0.22; 
		fbPIDDischrgCmdFromBackend.udiIValue := 450; 	
	ELSIF lrErrorPIDCorrectionDischrgCmdFromBackend > 2 AND lrErrorPIDCorrectionDischrgCmdFromBackend <= 2.5 THEN 
		fbPIDDischrgCmdFromBackend.rPValue := 0.26; 
		fbPIDDischrgCmdFromBackend.udiIValue := 675; 
	ELSIF lrErrorPIDCorrectionDischrgCmdFromBackend > 2.5 AND lrErrorPIDCorrectionDischrgCmdFromBackend <= 3 THEN 
		fbPIDDischrgCmdFromBackend.rPValue := 0.30; 
		fbPIDDischrgCmdFromBackend.udiIValue := 675;
	ELSIF lrErrorPIDCorrectionDischrgCmdFromBackend > 3 AND lrErrorPIDCorrectionDischrgCmdFromBackend <= 3.5 THEN 
		fbPIDDischrgCmdFromBackend.rPValue := 0.34; 
		fbPIDDischrgCmdFromBackend.udiIValue := 900;
	ELSIF lrErrorPIDCorrectionDischrgCmdFromBackend > 3.5 AND lrErrorPIDCorrectionDischrgCmdFromBackend <= 4 THEN 
		fbPIDDischrgCmdFromBackend.rPValue := 0.38; 
		fbPIDDischrgCmdFromBackend.udiIValue := 900;
	ELSIF lrErrorPIDCorrectionDischrgCmdFromBackend > 4 AND lrErrorPIDCorrectionDischrgCmdFromBackend <= 4.5 THEN 
		fbPIDDischrgCmdFromBackend.rPValue := 0.42; 
		fbPIDDischrgCmdFromBackend.udiIValue := 900;
	ELSIF lrErrorPIDCorrectionDischrgCmdFromBackend > 4.5 AND lrErrorPIDCorrectionDischrgCmdFromBackend <= 5 THEN 
		fbPIDDischrgCmdFromBackend.rPValue := 0.46; 
		fbPIDDischrgCmdFromBackend.udiIValue := 900;
	ELSIF lrErrorPIDCorrectionDischrgCmdFromBackend > 5 THEN 
		fbPIDDischrgCmdFromBackend.rPValue := 0.50; 
		fbPIDDischrgCmdFromBackend.udiIValue := 900;
	END_IF
ELSIF eSpeedModeBackendController = E_SpeedModeBackendController_EMS.eFast THEN
	IF lrErrorPIDCorrectionDischrgCmdFromBackend <= 0.5 THEN 
		fbPIDDischrgCmdFromBackend.rPValue := 0.40; 
		fbPIDDischrgCmdFromBackend.udiIValue := 275;
	ELSIF lrErrorPIDCorrectionDischrgCmdFromBackend > 0.5 AND lrErrorPIDCorrectionDischrgCmdFromBackend <= 1 THEN 
		fbPIDDischrgCmdFromBackend.rPValue := 0.42; 
		fbPIDDischrgCmdFromBackend.udiIValue := 275;
	ELSIF lrErrorPIDCorrectionDischrgCmdFromBackend > 1 AND lrErrorPIDCorrectionDischrgCmdFromBackend <= 1.5 THEN 
		fbPIDDischrgCmdFromBackend.rPValue := 0.44; 
		fbPIDDischrgCmdFromBackend.udiIValue := 275; 
	ELSIF lrErrorPIDCorrectionDischrgCmdFromBackend > 1.5 AND lrErrorPIDCorrectionDischrgCmdFromBackend <= 2 THEN 
		fbPIDDischrgCmdFromBackend.rPValue := 0.46; 
		fbPIDDischrgCmdFromBackend.udiIValue := 275; 	
	ELSIF lrErrorPIDCorrectionDischrgCmdFromBackend > 2 AND lrErrorPIDCorrectionDischrgCmdFromBackend <= 2.5 THEN 
		fbPIDDischrgCmdFromBackend.rPValue := 0.48; 
		fbPIDDischrgCmdFromBackend.udiIValue := 500; 
	ELSIF lrErrorPIDCorrectionDischrgCmdFromBackend > 2.5 AND lrErrorPIDCorrectionDischrgCmdFromBackend <= 3 THEN 
		fbPIDDischrgCmdFromBackend.rPValue := 0.50; 
		fbPIDDischrgCmdFromBackend.udiIValue := 500;
	ELSIF lrErrorPIDCorrectionDischrgCmdFromBackend > 3 AND lrErrorPIDCorrectionDischrgCmdFromBackend <= 3.5 THEN 
		fbPIDDischrgCmdFromBackend.rPValue := 0.52; 
		fbPIDDischrgCmdFromBackend.udiIValue := 750;
	ELSIF lrErrorPIDCorrectionDischrgCmdFromBackend > 3.5 AND lrErrorPIDCorrectionDischrgCmdFromBackend <= 4 THEN 
		fbPIDDischrgCmdFromBackend.rPValue := 0.54; 
		fbPIDDischrgCmdFromBackend.udiIValue := 750;
	ELSIF lrErrorPIDCorrectionDischrgCmdFromBackend > 4 AND lrErrorPIDCorrectionDischrgCmdFromBackend <= 4.5 THEN 
		fbPIDDischrgCmdFromBackend.rPValue := 0.56; 
		fbPIDDischrgCmdFromBackend.udiIValue := 750;
	ELSIF lrErrorPIDCorrectionDischrgCmdFromBackend > 4.5 AND lrErrorPIDCorrectionDischrgCmdFromBackend <= 5 THEN 
		fbPIDDischrgCmdFromBackend.rPValue := 0.58; 
		fbPIDDischrgCmdFromBackend.udiIValue := 750;
	ELSIF lrErrorPIDCorrectionDischrgCmdFromBackend > 5 THEN 
		fbPIDDischrgCmdFromBackend.rPValue := 0.60; 
		fbPIDDischrgCmdFromBackend.udiIValue := 750;
	END_IF
END_IF

fbPIDDischrgCmdFromBackend(
	bEnable:= , 
	rSetpoint:= LREAL_TO_REAL(lrNewBatteryPowerWithCorrection), 
	udiIValue:= , 
	udiDValue:= 0, 
	udiDamping:= 0, 
	rPValue:= , 
	rMaxValue:= 100, 
	rMinValue:= 0,
	rNeutralZone:= 0.1, 
	bDirection:= FALSE, 
	rActualValue:= LREAL_TO_REAL(lrActualPowerBatterys), 
	rQController=> rControllerQPIDDischrgCmdFromBackend);

IF eOperationMode = E_OperatingMode_EMS.eSelfConsumption THEN 
	FOR liLPDischrgCmdFromBackend := 1 TO Constants_Energy.diMaxNumberOfBatteryInverters BY 1 DO
		IF Lynus_Standards.GVL_Energy.stDataOfBatteryInverters[diNrOfEMS_OUT,liLPDischrgCmdFromBackend].byPriority <> 0 AND NOT bEPMActive AND bDischrgCmdFromBackendOK AND	
		arrMinPrioReached[1] AND arrMinPrioReached[2] AND arrMinPrioReached[3] AND arrMinPrioReached[4] AND arrMinPrioReached[5] THEN
			Lynus_Standards.GVL_Energy.stDataOfBatteryInverters[diNrOfEMS_OUT,liLPDischrgCmdFromBackend].rTargetPowerEMS := rControllerQPIDDischrgCmdFromBackend;
		END_IF 
	END_FOR	
ELSE
	FOR liLPDischrgCmdFromBackend := 1 TO Constants_Energy.diMaxNumberOfBatteryInverters BY 1 DO
		IF Lynus_Standards.GVL_Energy.stDataOfBatteryInverters[diNrOfEMS_OUT,liLPDischrgCmdFromBackend].byPriority <> 0 AND NOT bEPMActive AND fbPIDDischrgCmdFromBackend.bEnable THEN
			Lynus_Standards.GVL_Energy.stDataOfBatteryInverters[diNrOfEMS_OUT,liLPDischrgCmdFromBackend].rTargetPowerEMS := rControllerQPIDDischrgCmdFromBackend;
		END_IF 
	END_FOR	
END_IF

//On this Modes set the Battery Power to 0 when no charge and no discharge controller is active
IF eOperationMode = E_OperatingMode_EMS.eLoadManagement OR eOperationMode = E_OperatingMode_EMS.ePeakLoadCapping THEN
	IF NOT fbPIDBatteryPLCLM_Chrg.bEnable AND NOT fbPIDBatteryPLCLM_Dischrg.bEnable AND NOT fbPIDDischrgCmdFromBackend.bEnable THEN
		FOR liLPDischrgCmdFromBackend := 1 TO Constants_Energy.diMaxNumberOfBatteryInverters BY 1 DO
			Lynus_Standards.GVL_Energy.stDataOfBatteryInverters[diNrOfEMS_OUT,liLPDischrgCmdFromBackend].rTargetPowerEMS := 0;
		END_FOR	
	END_IF
END_IF	    

(*------------------------------------------------------------------------------Progress and State----------------------------------------------------------------------------------------*)
	
IF NOT arrMinPrioReached[1] AND NOT arrMinPrioReached[2] AND NOT arrMinPrioReached[3] AND NOT arrMinPrioReached[4] AND NOT arrMinPrioReached[5] THEN
	byProgress := REAL_TO_BYTE(F_Scalvalue(x:= UINT_TO_REAL(uiState), x1:= 0, y1:= 0, x2:= 110, y2:= 100));
ELSE
	byProgress := 100;
END_IF 
byProgress := LIMIT(0,byProgress,100);

uiState_OUT := uiState;
	
(*-----------------------------------------------------------Write data to Global structure for batterys and battery inverters-----------------------------------------------------------------*)

FOR liLPBatterysSetupData := 1 TO Constants_Energy.diMaxNumberOfBatteryInverters BY 1 DO
	Lynus_Standards.GVL_Energy.stDataOfBatteryInverters[diNrOfEMS_OUT,liLPBatterysSetupData].byReserveSOCEPO := stSetupEMS.byReserveSOCEPO;
	Lynus_Standards.GVL_Energy.stDataOfBatteryInverters[diNrOfEMS_OUT,liLPBatterysSetupData].byMaxDepthOfDischargeEPO := stSetupEMS.byMaxDepthOfDischrgEPO;	
END_FOR

(*----------------------------------------------------------Handle messages from this device-----------------------------------------------------------------*)

fbMessagesEMS.wMessageCode := 0;

IF arrMinPrioReached[1] AND arrMinPrioReached[2] AND arrMinPrioReached[3] AND arrMinPrioReached[4] AND arrMinPrioReached[5] THEN 
	fbMessagesEMS.wMessageCode := 1; 
END_IF
IF arrMaxPrioReached[1] AND arrMaxPrioReached[2] AND arrMaxPrioReached[3] AND arrMaxPrioReached[4] AND arrMaxPrioReached[5] THEN 
	fbMessagesEMS.wMessageCode := 2;
END_IF
IF bMissingPowerData THEN 
	fbMessagesEMS.wMessageCode := 3; 
END_IF
IF bStopAll THEN 
	fbMessagesEMS.wMessageCode := 4; 
END_IF
IF bStopAll AND timDissableFunctions.Q THEN 
	fbMessagesEMS.wMessageCode := 5; 
END_IF

fbMessagesEMS(bEnable:= bEnable, wMessageCode:= , eMessageEMS=> eMessageEMS);

(*----------------------------------------------------------Save persistent data----------------------------------------------------------------*)

arrPD[1](lrValue:= BOOL_TO_LREAL(bEnable), bEventBasedActive=> );
arrPD[2](lrValue:= DINT_TO_LREAL(diNrOfEM_IN_ECS), bEventBasedActive=> );
arrPD[3](lrValue:= BYTE_TO_LREAL(stSetupEMS.byReserveSOCEPO), bEventBasedActive=> );
arrPD[4](lrValue:= BYTE_TO_LREAL(stSetupEMS.byMaxDepthOfDischrgEPO), bEventBasedActive=> );
arrPD[5](lrValue:= BYTE_TO_LREAL(stSetupEMS.byResChrgfromGridToBatt), bEventBasedActive=> );
arrPD[6](lrValue:= INT_TO_LREAL(eOperationMode), bEventBasedActive=> );
arrPD[7](lrValue:= REAL_TO_LREAL(stSetupEMS.rSizeMainFuseCS), bEventBasedActive=> );
arrPD[8](lrValue:= UINT_TO_LREAL(stSetupEMS.uiUpdateTime), bEventBasedActive=> );
arrPD[9](lrValue:= INT_TO_LREAL(eSpeedModeBackendController), bEventBasedActive=> );
arrPD[10](lrValue:= BOOL_TO_LREAL(stSetupEMS.bAllowChrgFromGrid), bEventBasedActive=> );
arrPD[11](lrValue:= BOOL_TO_LREAL(stSetupEMS.bEnableMainFuseFunction), bEventBasedActive=> );
arrPD[12](lrValue:= BYTE_TO_LREAL(stSetupEMS.byPrioMinChrgBattSOCInEPO), bEventBasedActive=> );

(*----------------------------------------------------------impuls for start/stop charging battery----------------------------------------------------------------*)
IF b_EnableBatteryChargingControl THEN
	IF b_StartReleaseBatteryCharging THEN // AND NOT b_StopReleaseBatteryCharging THEN
		RS_BatteryChargingControl.SET:=TRUE;
		RS_BatteryChargingControl.RESET1:=FALSE;
	ELSIF NOT b_StartReleaseBatteryCharging AND b_StopReleaseBatteryCharging THEN
			RS_BatteryChargingControl.SET:=FALSE;
		RS_BatteryChargingControl.RESET1:=TRUE;
	END_IF
ELSE
	RS_BatteryChargingControl.RESET1:=TRUE;
	RS_BatteryChargingControl.SET:=false;
END_IF

RS_BatteryChargingControl(Q1=>b_TimeBasedReleaseChargingBattery);

END_FUNCTION_BLOCK

// ---- POUs/prgCS.TcPOU
PROGRAM prgCS
VAR PERSISTENT
	bEnabledCS				: BOOL;									//{#lynus.ag#()}
	byPrioCS				: BYTE;									//{#lynus.ag#()}
	bySOC_E_CS				: BYTE;									//{#lynus.ag#()}
	bySOC_D_CS				: BYTE;									//{#lynus.ag#()}
	byMinPowerCS			: BYTE;									//{#lynus.ag#()}
	rMaxPowerCS				: REAL;									//{#lynus.ag#()}
END_VAR
VAR
	fbCS					: FB_ECS_Alpitronic_Hypercharger;
	bIsEnabledCS			: BOOL;									//{#lynus.ag#()}
	byErrorWarningCS		: BYTE;									//{#lynus.ag#()}
	byStateMinPowerCS		: BYTE;									//{#lynus.ag#()}
	rTargetPowerCS			: REAL;									//{#lynus.ag#()}
	bCarConnected			: BOOL;									//{#lynus.ag#()}
	rChrgTime				: REAL;									//{#lynus.ag#()}
	lrPowerCS				: LREAL;								//{#lynus.ag#()}
END_VAR

fbCS.stSetupECS.byDisableSOC := bySOC_D_CS;
	fbCS.stSetupECS.byEnableSOC := bySOC_E_CS;
		fbCS.stSetupECS.byPriority := byPrioCS;
			fbCS.stSetupECS.rMaxPower := rMaxPowerCS;
				fbCS.stSetupECS.byCSMinPower := byMinPowerCS;

fbCS(
	bEnable:= bEnabledCS, 
	bPowerDataInvers:= , 
	byUnitID:= 1,									// Always 1 
	diNrOfEMS_IN:= prgEMS.fbEMS.diNrOfEMS_OUT, 
	diNrOfEM_IN_CS:= , 
	sIPAdress:= '192.168.1.101', 						// modify IP Adress
	stSetupECS:= , 
	stDataECS=> , 
	diNrOfECS_OUT=> );

bIsEnabledCS := fbCS.stDataECS.bEnabled;
	byStateMinPowerCS := fbCS.stDataECS.bySCSMinPower;
		rTargetPowerCS := fbCS.stDataECS.rTargetPower;	
			byErrorWarningCS := fbCS.stDataECS.byErrorWarning;
				bCarConnected := fbCS.stDataECS.bCarConnected;
					rChrgTime := fbCS.stDataECS.arrChargingTimeInMin[1];
						lrPowerCS := fbCS.stDataECS.lrTotalPower;

END_PROGRAM

// ---- POUs/prgGrid.TcPOU
PROGRAM prgGrid
VAR PERSISTENT
	rSizeGridConn				: REAL;									//{#lynus.ag#()}
	lrCounterGridProd			: LREAL;								//{#lynus.ag#()}
	lrCounterGridCons			: LREAL;								//{#lynus.ag#()}
END_VAR
VAR
	fbGrid						: FB_Grid_Power;
	fbGridCounter				: FB_EnergyCounter;
	lrGridPower					: LREAL;								//{#lynus.ag#()}
END_VAR

fbGrid(
	bEnable:= TRUE, 
	diNrOfEMS_IN:= prgEMS.fbEMS.diNrOfEMS_OUT, 
	diNrOfEM_IN_Grid:= prgEM.fbEM1.diNrOfEM_OUT, 
	rSizeGridConn:= rSizeGridConn, 
	stDataGrid=> , 
	diNrOfGrid_OUT=> );
	
lrGridPower := fbGrid.stDataGrid.lrPower;


// EnergyCounter
fbGridCounter(
	byActiveTariff:= 1, 
	lrPowerInput:= lrGridPower, 
	lrTotalCounterEnergy_Consumption=> , 
	lrTotalCounterEnergy_Production=> , 
	lrCounterEnergyT1_Consumption=> , 
	lrCounterEnergyT2_Consumption=> , 
	lrCounterEnergyT1_Production=> , 
	lrCounterEnergyT2_Production=> );

	IF fbGridCounter.lrTotalCounterEnergy_Production > lrCounterGridProd THEN  	
			lrCounterGridProd := fbGridCounter.lrTotalCounterEnergy_Production;
	END_IF

		IF fbGridCounter.lrTotalCounterEnergy_Consumption > lrCounterGridCons THEN  	
			lrCounterGridCons := fbGridCounter.lrTotalCounterEnergy_Consumption;
		END_IF

END_PROGRAM

// ---- POUs/prgEM.TcPOU
PROGRAM prgEM
VAR
	fbKBusState		: FB_K_Bus_State;
	fbEM1			: FB_EM_Beckhoff_KL3403;
	bGridEnabled	: BOOL;								//{#lynus.ag#()}
	lrPowerGrid		: LREAL;							//{#lynus.ag#()}
	lrPowerEM1_1	: LREAL;							//{#lynus.ag#()}
	lrPowerEM1_2	: LREAL;							//{#lynus.ag#()}
	lrPowerEM1_3	: LREAL;							//{#lynus.ag#()}
	lr_GridVoltageL1N_V			: LREAL;							//{#lynus.ag#()}
	lr_GridVoltageL2N_V			: LREAL;							//{#lynus.ag#()}
	lr_GridVoltageL3N_V			: LREAL;							//{#lynus.ag#()}

	lrReactivePowerGrid			: LREAL;							//{#lynus.ag#()}
	lrApparentPowerGrid			: LREAL;							//{#lynus.ag#()}

	r_PF1: REAL;
	r_PF2: REAL;
	r_PF3: REAL;
	r_Current1: REAL;
	r_Current2: REAL;
	r_Current3: REAL;
END_VAR
VAR PERSISTENT
END_VAR

//The mapping of this function must be linked with the K-Bus State in the E/A Part
fbKBusState(	uiKBusState_OUT=> , 
				b_Kbus_notOk=> , 
				word_ErrorCount=> );
				
//The mapping of this function must be linked with the KL3403 in the E/A Part
//UV1
fbEM1(
	bEnable:= TRUE, 
	bChannel1Invers:= FALSE,				//Invert power data when transformer are mounted upside down
	bChannel2Invers:= FALSE,
	bChannel3Invers:= FALSE,
	uiCurrentTransformerRatioL1:= 400, //Transformer ratio on the secondary side
	uiCurrentTransformerRatioL2:= 400, 
	uiCurrentTransformerRatioL3:= 400, 
	uiKBusState_IN:= fbKBusState.uiKBusState_OUT, 
	stDataEMPower=> , 
	stDataEMCounter=> , 
	stDataEMPowerRealTime=> , 
	stDataEMCounterRealTime=> , 
	diNrOfEM_OUT=> );

lrPowerGrid := fbEM1.stDataEMPower.lrPowerTotal;	
lrPowerEM1_1 := fbEM1.stDataEMPower.lrPowerL1;
lrPowerEM1_2 := fbEM1.stDataEMPower.lrPowerL2;
lrPowerEM1_3 := fbEM1.stDataEMPower.lrPowerL3;
bGridEnabled := fbEM1.bEnable;
					
					
lrReactivePowerGrid:=fbEM1.stDataEMPower.lrReactivePowerTotal;
lrApparentPowerGrid:=fbEM1.stDataEMPower.lrApparentPowerTotal;

lr_GridVoltageL1N_V:=fbEM1.stDataEMPower.lrVoltageL1N;
lr_GridVoltageL2N_V:=fbEM1.stDataEMPower.lrVoltageL2N;
lr_GridVoltageL3N_V:=fbEM1.stDataEMPower.lrVoltageL3N;

r_PF1 := fbem1.stDataL1.rPowerfactor;
r_PF2 := fbem1.stDataL2.rPowerfactor;
r_PF3 := fbem1.stDataL3.rPowerfactor;

r_Current1 := fbem1.stDataL1.rCurrent;
r_Current2 := fbem1.stDataL2.rCurrent;
r_Current3 := fbem1.stDataL3.rCurrent;

END_PROGRAM

// ---- POUs/prgHouse.TcPOU
PROGRAM prgHouse
VAR
	fbHouse				: FB_HouseC_Power_Virtual;
	bHouseEnabled		: BOOL;						//{#lynus.ag#()}
	lrPowerHouse		: LREAL;					//{#lynus.ag#()}
END_VAR
VAR PERSISTENT
	bEnableHouse		: BOOL;						//{#lynus.ag#()}
END_VAR

fbHouse(
	bEnable:= bEnableHouse, 
	diNrOfEMS_IN:= prgEMS.fbEMS.diNrOfEMS_OUT, 
	bSetDefault:= , 
	lrCounterConsumptionSetDefault:= , 
	lrCounterProductionSetDefault:= , 
	stDataHouseC=> , 
	diNrOfHouseC_OUT=> );
	
bHouseEnabled := fbHouse.stDataHouseC.bEnabled;
	lrPowerHouse := fbHouse.stDataHouseC.lrPower-prgCS.lrPowerCS;

END_PROGRAM

// ---- POUs/prgPV.TcPOU
PROGRAM prgPV
VAR
	fbPV					: FB_Symo_PV_Inverter_FLOAT_1_DM_30_Inverter;
	fbPVInt					: FB_PV_Power;
	fbPVCounter				: FB_EnergyCounter;
	lrPowerPV				: LREAL;				//{#lynus.ag#()}
	byErrorWarningPV		: BYTE;					//{#lynus.ag#()}
	
	// extend or reduce amount of PV Inverters
	lrPowerPV_1				: LREAL;				//{#lynus.ag#()}
	lrPowerPV_2				: LREAL;				//{#lynus.ag#()}
	lrPowerPV_3				: LREAL;				//{#lynus.ag#()}
	lrPowerPV_4				: LREAL;				//{#lynus.ag#()}
END_VAR
VAR PERSISTENT
	lrCounterPV				: LREAL;				//{#lynus.ag#()}
END_VAR

// extend or reduce amount of PV Inverters
fbPV.arrUnitID_Inverter[1] := 1;
fbPV.arrUnitID_Inverter[2] := 2;
fbPV.arrUnitID_Inverter[3] := 3;
fbPV.arrUnitID_Inverter[4] := 4;

fbPV(
	bEnable:= TRUE, 
	sIPAdress:= '192.168.1.100', 			// modify IP Adress
	arrUnitID_Inverter:= , 
	arrDataSymo10=> , 
	stDataEMPower_PV=> , 
	stDataEMCounter_PV=> , 
	diNrOfEM_OUT_PV=> );

// extend or reduce amount of PV Inverters
lrPowerPV_1 := fbPV.arrDataSymo10[1].lrPowerAcInverter;
lrPowerPV_2 := fbPV.arrDataSymo10[2].lrPowerAcInverter;
lrPowerPV_3 := fbPV.arrDataSymo10[3].lrPowerAcInverter;
lrPowerPV_4 := fbPV.arrDataSymo10[4].lrPowerAcInverter;
	
fbPVInt(
	bEnable:= TRUE, 
	bPowerDataInvers:= , 
	diNrOfEM_IN_PV:= fbPV.diNrOfEM_OUT_PV, 
	stDataPv=> , 
	diNrOfPv_OUT=> );
	
lrPowerPV := fbPVInt.stDataPv.lrPower;
	byErrorWarningPV := fbPVInt.stDataPv.byErrorWarning;

// EnergyCounter
fbPVCounter(
	byActiveTariff:= 1, 
	lrPowerInput:= 0 - lrPowerPV, 
	lrTotalCounterEnergy_Consumption=> , 
	lrTotalCounterEnergy_Production=> , 
	lrCounterEnergyT1_Consumption=> , 
	lrCounterEnergyT2_Consumption=> , 
	lrCounterEnergyT1_Production=> , 
	lrCounterEnergyT2_Production=> );
	
IF fbPVCounter.lrTotalCounterEnergy_Production > lrCounterPV THEN  	
	lrCounterPV := fbPVCounter.lrTotalCounterEnergy_Production;
END_IF

END_PROGRAM

// ---- POUs/prgComEffIO.TcPOU
PROGRAM prgComEffIO
VAR
	fbCom		: FB_MqttCommunicator_V3;
END_VAR

fbCom(
	bConnect:= TRUE, 
	strAuthKey:=  'BMS99299754422' , 
	sUserName:= '673dfecd-87ae-41b4-adc6-bf4a9ec1d31b', 
	sUserPassword:= '6bd7bf44-8c7f-4537-ab63-8e71aabc2a94', 
	eSavePositionCertificate:= eSavePositionOnPLC.ePostionHardDisk, 
	time_HeartBeat_sec := T#15S,
	bConnected=> , 
	bError=> , 
	hrErrorCode=> , 
	eConnectionState=> , 
	eErrorMessage_Out=> );
	
(*old 
	sUserName:= '21f91cb5-8a07-4d3e-84c2-8bec390be0dd', 
	sUserPassword:= '26145dc9-e42c-4011-8f9c-6df6dcfb29f6', 
*)

END_PROGRAM

